// TIA Portal V20 export
FUNCTION_BLOCK "CallInterfaceSignals"   // FB38, LAD
TITLE = CallInterfaceSignals
AUTHOR : SICAR
FAMILY : Diag
VERSION : 1.0
// Der Baustein dient als Aufrufschnittstelle für den Funktionsbaustein „LSicar_InterfaceSignalsBool“. Er ist als Funktionsbaustein ausgeführt, um die intern aufgerufenen FBs mittels Multiinstanzen realisieren zu können.  
// Die Funktionsbausteine und das zugehörige WinCC-Bild sind für 16 Signaldatensätze („Schnittstelle Signale 01“ … „Schnittstellen Signale 16“) mit jeweils 32 boolschen Signalen vorgesehen.  
// 
// **PLC-Datentypen**  
//  LSicar_typeInterfaceSignalsBool 
//  typeInterfaceSignalsHmi 
//  LSicar _typeInterfaceSignals 
// 
// **WinCC-Diagnosebild**  
// 
// ![Icon](_Icon/reference.PNG)
// 
// siehe ..\Library Types\LSicar_InterfaceSignalsBool.pdf  
// 
//  
// 
// **Beispielaufruf**  
// Abbildung in Kontaktplan (KOP).  D:\Software\Symbols_Icons\BMPs-JPGs-PNGs\Verschiedene\symb_user_goto_transparent.pngEin lauffähiger Programm-Aufruf hierzu ist im „SICAR-StartUp“-Projekt enthalten.  
// 
// **Aufrufschnittstelle**  
// Der Baustein wird einmalig im zyklischen Programm aufgerufen.  
// 
// **Intern verwendete „Erweiterte Anweisungen / Bausteine“**  
// ..\Library Types\LSicar_InterfaceSignalsBool.pdf
// The block serves as a calling interface of the block “InterfaceSignalsBool“. The block is designed as function block in order to implement the block calls as multi-instances.
// stored: IsIECCheckEnabled true, MemoryReserve 100, SetENOAutomatically true
   VAR
      statReadValueHmi : Bool;   // HMI: Lese Signalwert / HMI: Read value signal
      statSelectSignalsHmi : USInt := 1;   // HMI: Angewählte Interface Schnittstelle (1..16) / HMI: Selected interface signals (1..16)
      statSelectSignalsOld { ExternalAccessible := 'False'; ExternalVisible := 'False'; ExternalWritable := 'False'} : USInt;   // Altwert: Angewählte Interface Schnittstelle / Old value: Selected interface signals
      statRisEdgeReadName { ExternalAccessible := 'False'; ExternalVisible := 'False'; ExternalWritable := 'False'} : Bool;   // Steigende Flanke / Rising edge
      statPosPulseReadName : Bool;   // Positiver Impuls / Positive pulse
      statInterfaceSignalsHmi : Array[0..99] of "typeInterfaceSignalsHmi";   // HMI: Beschreibung, Wert und Symbolischer Name / HMI: Description, value and symbolic name
      instSignals1Left { S7_SetPoint := 'True'} : "LAF_InterfaceSignalsBool";
      instSignals1Right { S7_SetPoint := 'True'} : "LAF_InterfaceSignalsBool";
      instSignals2Left { S7_SetPoint := 'True'} : "LAF_InterfaceSignalsBool";
      instSignals2Right { S7_SetPoint := 'True'} : "LAF_InterfaceSignalsBool";
      instSignals3Left { S7_SetPoint := 'True'} : "LAF_InterfaceSignalsBool";
      instSignals3Right { S7_SetPoint := 'True'} : "LAF_InterfaceSignalsBool";
      instSignals4Left { S7_SetPoint := 'True'} : "LAF_InterfaceSignalsBool";
      instSignals4Right { S7_SetPoint := 'True'} : "LAF_InterfaceSignalsBool";
      instSignals5Left { S7_SetPoint := 'True'} : "LAF_InterfaceSignalsBool";
      instSignals5Right { S7_SetPoint := 'True'} : "LAF_InterfaceSignalsBool";
      instSignals6Left { S7_SetPoint := 'True'} : "LAF_InterfaceSignalsBool";
      instSignals6Right { S7_SetPoint := 'True'} : "LAF_InterfaceSignalsBool";
      instSignals7Left { S7_SetPoint := 'True'} : "LAF_InterfaceSignalsBool";
      instSignals7Right { S7_SetPoint := 'True'} : "LAF_InterfaceSignalsBool";
      instSignals8Left { S7_SetPoint := 'True'} : "LAF_InterfaceSignalsBool";
      instSignals8Right { S7_SetPoint := 'True'} : "LAF_InterfaceSignalsBool";
      instSignals9Left { S7_SetPoint := 'True'} : "LAF_InterfaceSignalsBool";
      instSignals9Right { S7_SetPoint := 'True'} : "LAF_InterfaceSignalsBool";
      instSignals10Left { S7_SetPoint := 'True'} : "LAF_InterfaceSignalsBool";
      instSignals10Right { S7_SetPoint := 'True'} : "LAF_InterfaceSignalsBool";
      instSignals11Left { S7_SetPoint := 'True'} : "LAF_InterfaceSignalsBool";
      instSignals11Right { S7_SetPoint := 'True'} : "LAF_InterfaceSignalsBool";
      instSignals12Left { S7_SetPoint := 'True'} : "LAF_InterfaceSignalsBool";
      instSignals12Right { S7_SetPoint := 'True'} : "LAF_InterfaceSignalsBool";
      instSignals13Left { S7_SetPoint := 'True'} : "LAF_InterfaceSignalsBool";
      instSignals13Right { S7_SetPoint := 'True'} : "LAF_InterfaceSignalsBool";
      instSignals14Left { S7_SetPoint := 'True'} : "LAF_InterfaceSignalsBool";
      instSignals14Right { S7_SetPoint := 'True'} : "LAF_InterfaceSignalsBool";
      instSignals15Left { S7_SetPoint := 'True'} : "LAF_InterfaceSignalsBool";
      instSignals15Right { S7_SetPoint := 'True'} : "LAF_InterfaceSignalsBool";
      instSignals16Left { S7_SetPoint := 'True'} : "LAF_InterfaceSignalsBool";
      instSignals16Right { S7_SetPoint := 'True'} : "LAF_InterfaceSignalsBool";
      instSignals17Left { S7_SetPoint := 'True'} : "LAF_InterfaceSignalsBool";
      instSignals17Right { S7_SetPoint := 'True'} : "LAF_InterfaceSignalsBool";
      instSignals18Left { S7_SetPoint := 'True'} : "LAF_InterfaceSignalsBool";
      instSignals18Right { S7_SetPoint := 'True'} : "LAF_InterfaceSignalsBool";
      instSignals19Left { S7_SetPoint := 'True'} : "LAF_InterfaceSignalsBool";
      instSignals19Right { S7_SetPoint := 'True'} : "LAF_InterfaceSignalsBool";
      instSignals20Left { S7_SetPoint := 'True'} : "LAF_InterfaceSignalsBool";
      instSignals20Right { S7_SetPoint := 'True'} : "LAF_InterfaceSignalsBool";
      instSignals21Left { S7_SetPoint := 'True'} : "LAF_InterfaceSignalsBool";
      instSignals21Right { S7_SetPoint := 'True'} : "LAF_InterfaceSignalsBool";
      instSignals22Left { S7_SetPoint := 'True'} : "LAF_InterfaceSignalsBool";
      instSignals22Right { S7_SetPoint := 'True'} : "LAF_InterfaceSignalsBool";
      instSignals23Left { S7_SetPoint := 'True'} : "LAF_InterfaceSignalsBool";
      instSignals23Right { S7_SetPoint := 'True'} : "LAF_InterfaceSignalsBool";
      instSignals24Left { S7_SetPoint := 'True'} : "LAF_InterfaceSignalsBool";
      instSignals24Right { S7_SetPoint := 'True'} : "LAF_InterfaceSignalsBool";
      instSignals25Left { S7_SetPoint := 'True'} : "LAF_InterfaceSignalsBool";
      instSignals25Right { S7_SetPoint := 'True'} : "LAF_InterfaceSignalsBool";
      instSignals26Left { S7_SetPoint := 'True'} : "LAF_InterfaceSignalsBool";
      instSignals26Right { S7_SetPoint := 'True'} : "LAF_InterfaceSignalsBool";
      instSignals27Left { S7_SetPoint := 'True'} : "LAF_InterfaceSignalsBool";
      instSignals27Right { S7_SetPoint := 'True'} : "LAF_InterfaceSignalsBool";
      instSignals28Left { S7_SetPoint := 'True'} : "LAF_InterfaceSignalsBool";
      instSignals28Right { S7_SetPoint := 'True'} : "LAF_InterfaceSignalsBool";
      instSignals29Left { S7_SetPoint := 'True'} : "LAF_InterfaceSignalsBool";
      instSignals29Right { S7_SetPoint := 'True'} : "LAF_InterfaceSignalsBool";
      instSignals30Left { S7_SetPoint := 'True'} : "LAF_InterfaceSignalsBool";
      instSignals30Right { S7_SetPoint := 'True'} : "LAF_InterfaceSignalsBool";
      instSignals31Left { S7_SetPoint := 'True'} : "LAF_InterfaceSignalsBool";
      instSignals31Right { S7_SetPoint := 'True'} : "LAF_InterfaceSignalsBool";
      instSignals32Left { S7_SetPoint := 'True'} : "LAF_InterfaceSignalsBool";
      instSignals32Right { S7_SetPoint := 'True'} : "LAF_InterfaceSignalsBool";
      instSignals33Left { S7_SetPoint := 'True'} : "LAF_InterfaceSignalsBool";
      instSignals33Right { S7_SetPoint := 'True'} : "LAF_InterfaceSignalsBool";
      instSignals34Left { S7_SetPoint := 'True'} : "LAF_InterfaceSignalsBool";
      instSignals34Right { S7_SetPoint := 'True'} : "LAF_InterfaceSignalsBool";
      instSignals35Left { S7_SetPoint := 'True'} : "LAF_InterfaceSignalsBool";
      instSignals35Right { S7_SetPoint := 'True'} : "LAF_InterfaceSignalsBool";
      instSignals36Left { S7_SetPoint := 'True'} : "LAF_InterfaceSignalsBool";
      instSignals36Right { S7_SetPoint := 'True'} : "LAF_InterfaceSignalsBool";
      instSignals37Left { S7_SetPoint := 'True'} : "LAF_InterfaceSignalsBool";
      instSignals37Right { S7_SetPoint := 'True'} : "LAF_InterfaceSignalsBool";
      instSignals38Left { S7_SetPoint := 'True'} : "LAF_InterfaceSignalsBool";
      instSignals38Right { S7_SetPoint := 'True'} : "LAF_InterfaceSignalsBool";
      instSignals39Left { S7_SetPoint := 'True'} : "LAF_InterfaceSignalsBool";
      instSignals39Right { S7_SetPoint := 'True'} : "LAF_InterfaceSignalsBool";
      instSignals40Left { S7_SetPoint := 'True'} : "LAF_InterfaceSignalsBool";
      instSignals40Right { S7_SetPoint := 'True'} : "LAF_InterfaceSignalsBool";
      instSignals41Left { S7_SetPoint := 'True'} : "LAF_InterfaceSignalsBool";
      instSignals41Right { S7_SetPoint := 'True'} : "LAF_InterfaceSignalsBool";
      instSignals42Left { S7_SetPoint := 'True'} : "LAF_InterfaceSignalsBool";
      instSignals42Right { S7_SetPoint := 'True'} : "LAF_InterfaceSignalsBool";
      instSignals43Left { S7_SetPoint := 'True'} : "LAF_InterfaceSignalsBool";
      instSignals43Right { S7_SetPoint := 'True'} : "LAF_InterfaceSignalsBool";
      instSignals44Left { S7_SetPoint := 'True'} : "LAF_InterfaceSignalsBool";
      instSignals44Right { S7_SetPoint := 'True'} : "LAF_InterfaceSignalsBool";
      instSignals45Left { S7_SetPoint := 'True'} : "LAF_InterfaceSignalsBool";
      instSignals45Right { S7_SetPoint := 'True'} : "LAF_InterfaceSignalsBool";
      instSignals46Left { S7_SetPoint := 'True'} : "LAF_InterfaceSignalsBool";
      instSignals46Right { S7_SetPoint := 'True'} : "LAF_InterfaceSignalsBool";
      instSignals47Left { S7_SetPoint := 'True'} : "LAF_InterfaceSignalsBool";
      instSignals47Right { S7_SetPoint := 'True'} : "LAF_InterfaceSignalsBool";
      instSignals48Left { S7_SetPoint := 'True'} : "LAF_InterfaceSignalsBool";
      instSignals48Right { S7_SetPoint := 'True'} : "LAF_InterfaceSignalsBool";
      instSignals49Left { S7_SetPoint := 'True'} : "LAF_InterfaceSignalsBool";
      instSignals49Right { S7_SetPoint := 'True'} : "LAF_InterfaceSignalsBool";
      instSignals50Left { S7_SetPoint := 'True'} : "LAF_InterfaceSignalsBool";
      instSignals50Right { S7_SetPoint := 'True'} : "LAF_InterfaceSignalsBool";
      instSignals51Left { S7_SetPoint := 'True'} : "LAF_InterfaceSignalsBool";
      instSignals51Right { S7_SetPoint := 'True'} : "LAF_InterfaceSignalsBool";
      instSignals52Left { S7_SetPoint := 'True'} : "LAF_InterfaceSignalsBool";
      instSignals52Right { S7_SetPoint := 'True'} : "LAF_InterfaceSignalsBool";
      instSignals53Left { S7_SetPoint := 'True'} : "LAF_InterfaceSignalsBool";
      instSignals53Right { S7_SetPoint := 'True'} : "LAF_InterfaceSignalsBool";
      instSignals54Left { S7_SetPoint := 'True'} : "LAF_InterfaceSignalsBool";
      instSignals54Right { S7_SetPoint := 'True'} : "LAF_InterfaceSignalsBool";
      instSignals55Left { S7_SetPoint := 'True'} : "LAF_InterfaceSignalsBool";
      instSignals55Right { S7_SetPoint := 'True'} : "LAF_InterfaceSignalsBool";
      instSignals56Left { S7_SetPoint := 'True'} : "LAF_InterfaceSignalsBool";
      instSignals56Right { S7_SetPoint := 'True'} : "LAF_InterfaceSignalsBool";
      instSignals57Left { S7_SetPoint := 'True'} : "LAF_InterfaceSignalsBool";
      instSignals57Right { S7_SetPoint := 'True'} : "LAF_InterfaceSignalsBool";
      instSignals58Left { S7_SetPoint := 'True'} : "LAF_InterfaceSignalsBool";
      instSignals58Right { S7_SetPoint := 'True'} : "LAF_InterfaceSignalsBool";
      instSignals59Left { S7_SetPoint := 'True'} : "LAF_InterfaceSignalsBool";
      instSignals59Right { S7_SetPoint := 'True'} : "LAF_InterfaceSignalsBool";
      instSignals60Left { S7_SetPoint := 'True'} : "LAF_InterfaceSignalsBool";
      instSignals60Right { S7_SetPoint := 'True'} : "LAF_InterfaceSignalsBool";
      instSignals61Left { S7_SetPoint := 'True'} : "LAF_InterfaceSignalsBool";
      instSignals61Right { S7_SetPoint := 'True'} : "LAF_InterfaceSignalsBool";
      instSignals62Left { S7_SetPoint := 'True'} : "LAF_InterfaceSignalsBool";
      instSignals62Right { S7_SetPoint := 'True'} : "LAF_InterfaceSignalsBool";
      instSignals63Left { S7_SetPoint := 'True'} : "LAF_InterfaceSignalsBool";
      instSignals63Right { S7_SetPoint := 'True'} : "LAF_InterfaceSignalsBool";
      instSignals64Left { S7_SetPoint := 'True'} : "LAF_InterfaceSignalsBool";
      instSignals64Right { S7_SetPoint := 'True'} : "LAF_InterfaceSignalsBool";
      instSignals65Left { S7_SetPoint := 'True'} : "LAF_InterfaceSignalsBool";
      instSignals65Right { S7_SetPoint := 'True'} : "LAF_InterfaceSignalsBool";
      instSignals66Left { S7_SetPoint := 'True'} : "LAF_InterfaceSignalsBool";
      instSignals66Right { S7_SetPoint := 'True'} : "LAF_InterfaceSignalsBool";
      instSignals67Left { S7_SetPoint := 'True'} : "LAF_InterfaceSignalsBool";
      instSignals67Right { S7_SetPoint := 'True'} : "LAF_InterfaceSignalsBool";
      instSignals68Left { S7_SetPoint := 'True'} : "LAF_InterfaceSignalsBool";
      instSignals68Right { S7_SetPoint := 'True'} : "LAF_InterfaceSignalsBool";
      instSignals69Left { S7_SetPoint := 'True'} : "LAF_InterfaceSignalsBool";
      instSignals69Right { S7_SetPoint := 'True'} : "LAF_InterfaceSignalsBool";
      instSignals70Left { S7_SetPoint := 'True'} : "LAF_InterfaceSignalsBool";
      instSignals70Right { S7_SetPoint := 'True'} : "LAF_InterfaceSignalsBool";
      instSignals71Left { S7_SetPoint := 'True'} : "LAF_InterfaceSignalsBool";
      instSignals71Right { S7_SetPoint := 'True'} : "LAF_InterfaceSignalsBool";
      instSignals72Left { S7_SetPoint := 'True'} : "LAF_InterfaceSignalsBool";
      instSignals72Right { S7_SetPoint := 'True'} : "LAF_InterfaceSignalsBool";
      instSignals73Left { S7_SetPoint := 'True'} : "LAF_InterfaceSignalsBool";
      instSignals73Right { S7_SetPoint := 'True'} : "LAF_InterfaceSignalsBool";
      instSignals74Left { S7_SetPoint := 'True'} : "LAF_InterfaceSignalsBool";
      instSignals74Right { S7_SetPoint := 'True'} : "LAF_InterfaceSignalsBool";
      instSignals75Left { S7_SetPoint := 'True'} : "LAF_InterfaceSignalsBool";
      instSignals75Right { S7_SetPoint := 'True'} : "LAF_InterfaceSignalsBool";
      instSignals76Left { S7_SetPoint := 'True'} : "LAF_InterfaceSignalsBool";
      instSignals76Right { S7_SetPoint := 'True'} : "LAF_InterfaceSignalsBool";
      instSignals77Left { S7_SetPoint := 'True'} : "LAF_InterfaceSignalsBool";
      instSignals77Right { S7_SetPoint := 'True'} : "LAF_InterfaceSignalsBool";
      instSignals78Left { S7_SetPoint := 'True'} : "LAF_InterfaceSignalsBool";
      instSignals78Right { S7_SetPoint := 'True'} : "LAF_InterfaceSignalsBool";
      instSignals79Left { S7_SetPoint := 'True'} : "LAF_InterfaceSignalsBool";
      instSignals79Right { S7_SetPoint := 'True'} : "LAF_InterfaceSignalsBool";
      instSignals80Left { S7_SetPoint := 'True'} : "LAF_InterfaceSignalsBool";
      instSignals80Right { S7_SetPoint := 'True'} : "LAF_InterfaceSignalsBool";
      instSignals81Left { S7_SetPoint := 'True'} : "LAF_InterfaceSignalsBool";
      instSignals81Right { S7_SetPoint := 'True'} : "LAF_InterfaceSignalsBool";
      instSignals82Left { S7_SetPoint := 'True'} : "LAF_InterfaceSignalsBool";
      instSignals82Right { S7_SetPoint := 'True'} : "LAF_InterfaceSignalsBool";
      instSignals83Left { S7_SetPoint := 'True'} : "LAF_InterfaceSignalsBool";
      instSignals83Right { S7_SetPoint := 'True'} : "LAF_InterfaceSignalsBool";
      instSignals84Left { S7_SetPoint := 'True'} : "LAF_InterfaceSignalsBool";
      instSignals84Right { S7_SetPoint := 'True'} : "LAF_InterfaceSignalsBool";
      instSignals85Left { S7_SetPoint := 'True'} : "LAF_InterfaceSignalsBool";
      instSignals85Right { S7_SetPoint := 'True'} : "LAF_InterfaceSignalsBool";
      instSignals86Left { S7_SetPoint := 'True'} : "LAF_InterfaceSignalsBool";
      instSignals86Right { S7_SetPoint := 'True'} : "LAF_InterfaceSignalsBool";
      instSignals87Left { S7_SetPoint := 'True'} : "LAF_InterfaceSignalsBool";
      instSignals87Right { S7_SetPoint := 'True'} : "LAF_InterfaceSignalsBool";
      instSignals88Left { S7_SetPoint := 'True'} : "LAF_InterfaceSignalsBool";
      instSignals88Right { S7_SetPoint := 'True'} : "LAF_InterfaceSignalsBool";
      instSignals89Left { S7_SetPoint := 'True'} : "LAF_InterfaceSignalsBool";
      instSignals89Right { S7_SetPoint := 'True'} : "LAF_InterfaceSignalsBool";
      instSignals90Left { S7_SetPoint := 'True'} : "LAF_InterfaceSignalsBool";
      instSignals90Right { S7_SetPoint := 'True'} : "LAF_InterfaceSignalsBool";
      instSignals91Left { S7_SetPoint := 'True'} : "LAF_InterfaceSignalsBool";
      instSignals91Right { S7_SetPoint := 'True'} : "LAF_InterfaceSignalsBool";
      instSignals92Left { S7_SetPoint := 'True'} : "LAF_InterfaceSignalsBool";
      instSignals92Right { S7_SetPoint := 'True'} : "LAF_InterfaceSignalsBool";
      instSignals93Left { S7_SetPoint := 'True'} : "LAF_InterfaceSignalsBool";
      instSignals93Right { S7_SetPoint := 'True'} : "LAF_InterfaceSignalsBool";
      instSignals94Left { S7_SetPoint := 'True'} : "LAF_InterfaceSignalsBool";
      instSignals94Right { S7_SetPoint := 'True'} : "LAF_InterfaceSignalsBool";
      instSignals95Left { S7_SetPoint := 'True'} : "LAF_InterfaceSignalsBool";
      instSignals95Right { S7_SetPoint := 'True'} : "LAF_InterfaceSignalsBool";
      instSignals96Left { S7_SetPoint := 'True'} : "LAF_InterfaceSignalsBool";
      instSignals96Right { S7_SetPoint := 'True'} : "LAF_InterfaceSignalsBool";
      instSignals97Left { S7_SetPoint := 'True'} : "LAF_InterfaceSignalsBool";
      instSignals97Right { S7_SetPoint := 'True'} : "LAF_InterfaceSignalsBool";
      instSignals98Left { S7_SetPoint := 'True'} : "LAF_InterfaceSignalsBool";
      instSignals98Right { S7_SetPoint := 'True'} : "LAF_InterfaceSignalsBool";
      instSignals99Left { S7_SetPoint := 'True'} : "LAF_InterfaceSignalsBool";
      instSignals99Right { S7_SetPoint := 'True'} : "LAF_InterfaceSignalsBool";
   END_VAR
   VAR_TEMP
      tempLoopCounter : DInt;   // temp. Schleifenzähler / temp. Loop Counter
   END_VAR
   VAR_TEMP   // added for the SCL form of the ladder/FBD networks
      _w1 : Bool;
   END_VAR
BEGIN

REGION Network 1: Beschreibung / BLOCK INFO HEADER
   // **Betriebsart Automatik / Hand**  
   // Der Baustein ist keiner Betriebsart / Betriebsartenbereich zugeordnet.  
   // 
   // **Alarme**  
   // Der Baustein generiert keine Alarme.  
   // 
   // #### PLC-Datentypen  
   // Verwendete PLC-Datentypen für den SPS-Programmbaustein und das zugehörige WinCC-Bild.  
   // 
   // {.pageWidth}
   // ![Image](CallInterfaceSignals/de/image1.PNG)
   //  
   //  
   // #### Bausteinaufrufe 
   // Der Baustein “LSicar_InterfaceSignalsBool“ wird in diesem FB als Multi-Instanz aufgerufen, entspr. nebenstehender beispielhafter Darstellung.  
   // 
   // {.pageWidth}
   // ![Image](CallInterfaceSignals/de/image2.PNG)
   //  
   // Um einen neuen FB aufzurufen, ziehen Sie den FB in ein neues Netzwerk, wählen Sie „Multiinstanz“ aus, vergeben Sie einen Namen und parametrieren Sie den FB-Aufruf.  
   // 
   // {.pageWidth}
   // ![Image](CallInterfaceSignals/de/image3.PNG)
   //  
   //  
   // #### Weitere Hinweise 
   // 
   // #### Updateinfo 
   // 
   // #### Weitere Dokumente 
   // 
   // ![Icon](_Icon/reference.PNG)
   // 
   // ..\Library Types\LSicar_InterfaceSignalsBool.pdf
   // SIEMENS AG / (c)Copyright 2023
   // ------------------------------------------------------------------------------
   // Title:            CallInterfaceSignals (FB38)
   // Comment/Function: The block serves as a calling interface of the block “InterfaceSignalsBool“. The block is designed as function block in order to implement the block calls as multi-instances. 
   // Library/Family:   Diag
   // Author:           SICAR
   // Tested with:      ---
   // Engineering:      TIA Portal V19
   // Restrictions:     -
   // Requirements:     ---
   // ------------------------------------------------------------------------------
   // Change log table:
   // Version  | Date       | Expert in charge       | Changes applied
   // ---------|------------|------------------------|------------------------------
   // 01.00.00 | 11.12.2023 | SICAR
   //                         First released version
END_REGION

REGION Network 2: DESCRIPTION
   // Function block and corresponding WinCC screen are prepared for 16 data sets (“InterfaceSignals01“ through .”InterfaceSignals16“) with 32 Boolean signals each.  
   // 
   // **PLC-Data types**   
   // 
   // * LSicar_typeInterfaceSignalsBool 
   // * LSicar _typeInterfaceSignals 
   // * typeInterfaceSignalsHmi 
   // 
   // **WinCC-Faceplate**  
   // 
   // <None> 
   // 
   // **WinCC Diagnostic screen**   
   // 
   // See: ..\Library Types\LSicar_InterfaceSignalsBool.pdf  
   // 
   // **Block call example** 
   // 
   // View in ladder-logic (LAD), without parameter settings.  
   // An executable program call is available in the “SICAR-Startup” project.  
   // 
   // **Calling interface**  
   // 
   // The block is be called once in the cyclic program.  
   // 
   // **Internally used „Extended instructions / blocks“**  
   // 
   // See: ..\Library Types\LSicar_InterfaceSignalsBool.pdf
END_REGION

REGION Network 3: Initialisierung Loop_1 / Initialization Loop_1
   // Vorbesetzen des Schleifenindex / Preset the loop index
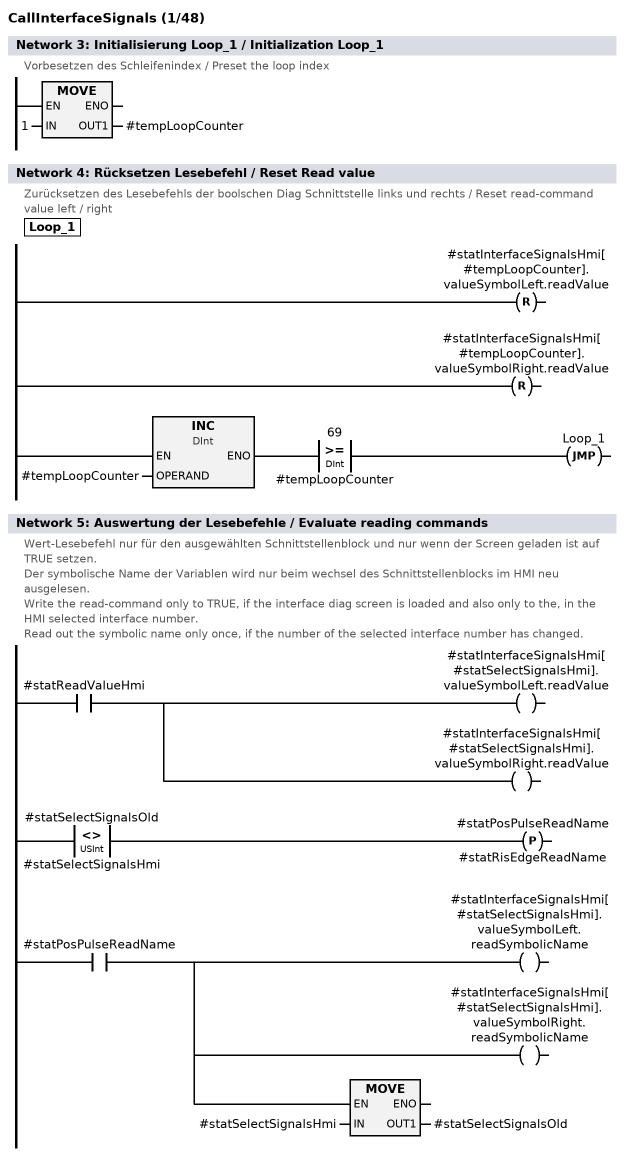
   RUNG wire#powerrail
      Move(in := 1, out1 => #tempLoopCounter)
   END_RUNG
   // the same network as SCL:
   #tempLoopCounter := 1;
END_REGION

REGION Network 4: Rücksetzen Lesebefehl / Reset Read value
   // Zurücksetzen des Lesebefehls der boolschen Diag Schnittstelle links und rechts / Reset read-command value left / right
   Label( Loop_1 )
   RUNG wire#powerrail
      R_Coil( #statInterfaceSignalsHmi[#tempLoopCounter].valueSymbolLeft.readValue )
   END_RUNG
   RUNG wire#powerrail
      R_Coil( #statInterfaceSignalsHmi[#tempLoopCounter].valueSymbolRight.readValue )
   END_RUNG
   RUNG wire#powerrail
      { S7_Templates := "DestType := DInt" } Inc( #tempLoopCounter )
      { S7_Templates := "SrcType := DInt" } GE_Contact(in1 := 69, in2 := #tempLoopCounter)
      JumpCoil( Loop_1 )
   END_RUNG
   // the same network as SCL:
   Loop_1:
   #statInterfaceSignalsHmi[#tempLoopCounter].valueSymbolLeft.readValue := FALSE;
   #statInterfaceSignalsHmi[#tempLoopCounter].valueSymbolRight.readValue := FALSE;
   #tempLoopCounter := #tempLoopCounter + 1;
   IF 69 >= #tempLoopCounter THEN GOTO Loop_1; END_IF;
END_REGION

REGION Network 5: Auswertung der Lesebefehle / Evaluate reading commands
   // Wert-Lesebefehl nur für den ausgewählten Schnittstellenblock und nur wenn der Screen geladen ist auf TRUE setzen.
   // Der symbolische Name der Variablen wird nur beim wechsel des Schnittstellenblocks im HMI neu ausgelesen.
   // Write the read-command only to TRUE, if the interface diag screen is loaded and also only to the, in the HMI selected interface number.
   // Read out the symbolic name only once, if the number of the selected interface number has changed.
   #statInterfaceSignalsHmi[#statSelectSignalsHmi].valueSymbolLeft.readValue := #statReadValueHmi;
   #statInterfaceSignalsHmi[#statSelectSignalsHmi].valueSymbolRight.readValue := #statReadValueHmi;
   #_w1 := #statSelectSignalsOld <> #statSelectSignalsHmi;
   #statPosPulseReadName := #_w1 AND NOT #statRisEdgeReadName;   // rising edge
   #statRisEdgeReadName := #_w1;
   #statInterfaceSignalsHmi[#statSelectSignalsHmi].valueSymbolLeft.readSymbolicName := #statPosPulseReadName;
   #statInterfaceSignalsHmi[#statSelectSignalsHmi].valueSymbolRight.readSymbolicName := #statPosPulseReadName;
   IF #statPosPulseReadName THEN #statSelectSignalsOld := #statSelectSignalsHmi; END_IF;
END_REGION

REGION Network 6: Interface Signals 03 -Example: System flags & Clock flags- / Interface Signals 01
   // Aufruf des Schnittstellen Signal Bausteins für die Systemvariablen / Call the interface signals bool blocks of system tags
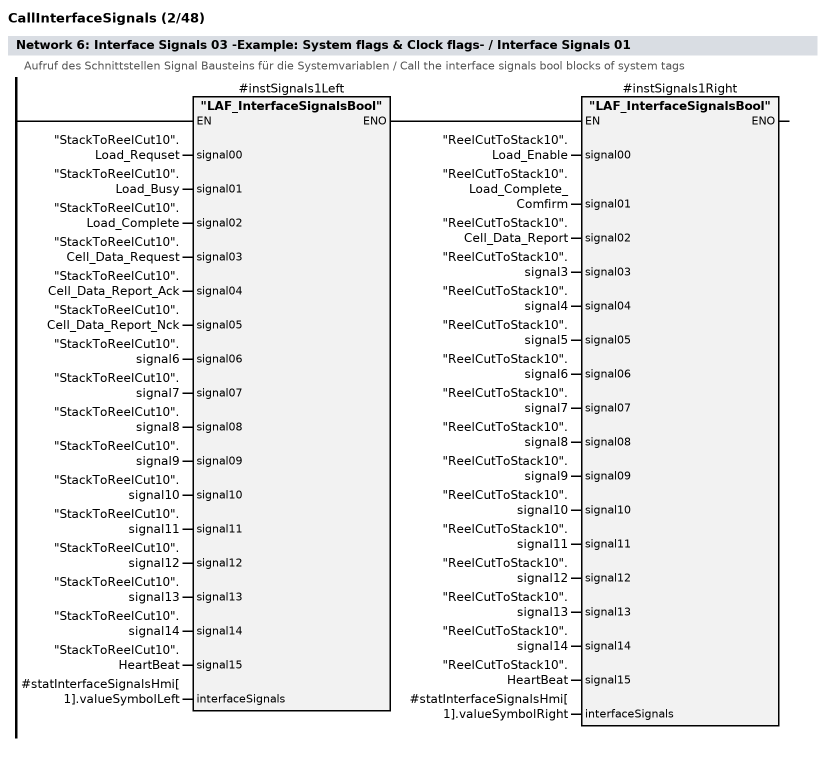
   RUNG wire#powerrail
      #instSignals1Left(signal00 := "StackToReelCut10".Load_Requset, signal01 := "StackToReelCut10".Load_Busy, signal02 := "StackToReelCut10".Load_Complete, signal03 := "StackToReelCut10".Cell_Data_Request, signal04 := "StackToReelCut10".Cell_Data_Report_Ack, signal05 := "StackToReelCut10".Cell_Data_Report_Nck, signal06 := "StackToReelCut10".signal6, signal07 := "StackToReelCut10".signal7, signal08 := "StackToReelCut10".signal8, signal09 := "StackToReelCut10".signal9, signal10 := "StackToReelCut10".signal10, signal11 := "StackToReelCut10".signal11, signal12 := "StackToReelCut10".signal12, signal13 := "StackToReelCut10".signal13, signal14 := "StackToReelCut10".signal14, signal15 := "StackToReelCut10".HeartBeat, interfaceSignals := #statInterfaceSignalsHmi[1].valueSymbolLeft)
      #instSignals1Right(signal00 := "ReelCutToStack10".Load_Enable, signal01 := "ReelCutToStack10".Load_Complete_Comfirm, signal02 := "ReelCutToStack10".Cell_Data_Report, signal03 := "ReelCutToStack10".signal3, signal04 := "ReelCutToStack10".signal4, signal05 := "ReelCutToStack10".signal5, signal06 := "ReelCutToStack10".signal6, signal07 := "ReelCutToStack10".signal7, signal08 := "ReelCutToStack10".signal8, signal09 := "ReelCutToStack10".signal9, signal10 := "ReelCutToStack10".signal10, signal11 := "ReelCutToStack10".signal11, signal12 := "ReelCutToStack10".signal12, signal13 := "ReelCutToStack10".signal13, signal14 := "ReelCutToStack10".signal14, signal15 := "ReelCutToStack10".HeartBeat, interfaceSignals := #statInterfaceSignalsHmi[1].valueSymbolRight)
   END_RUNG
   // the same network as SCL:
   #instSignals1Left(signal00 := "StackToReelCut10".Load_Requset,   // "LAF_InterfaceSignalsBool"
                     signal01 := "StackToReelCut10".Load_Busy,
                     signal02 := "StackToReelCut10".Load_Complete,
                     signal03 := "StackToReelCut10".Cell_Data_Request,
                     signal04 := "StackToReelCut10".Cell_Data_Report_Ack,
                     signal05 := "StackToReelCut10".Cell_Data_Report_Nck,
                     signal06 := "StackToReelCut10".signal6,
                     signal07 := "StackToReelCut10".signal7,
                     signal08 := "StackToReelCut10".signal8,
                     signal09 := "StackToReelCut10".signal9,
                     signal10 := "StackToReelCut10".signal10,
                     signal11 := "StackToReelCut10".signal11,
                     signal12 := "StackToReelCut10".signal12,
                     signal13 := "StackToReelCut10".signal13,
                     signal14 := "StackToReelCut10".signal14,
                     signal15 := "StackToReelCut10".HeartBeat,
                     interfaceSignals := #statInterfaceSignalsHmi[1].valueSymbolLeft,
                     ENO => #_w1);
   IF #_w1 THEN
       #instSignals1Right(signal00 := "ReelCutToStack10".Load_Enable,   // "LAF_InterfaceSignalsBool"
                          signal01 := "ReelCutToStack10".Load_Complete_Comfirm,
                          signal02 := "ReelCutToStack10".Cell_Data_Report,
                          signal03 := "ReelCutToStack10".signal3,
                          signal04 := "ReelCutToStack10".signal4,
                          signal05 := "ReelCutToStack10".signal5,
                          signal06 := "ReelCutToStack10".signal6,
                          signal07 := "ReelCutToStack10".signal7,
                          signal08 := "ReelCutToStack10".signal8,
                          signal09 := "ReelCutToStack10".signal9,
                          signal10 := "ReelCutToStack10".signal10,
                          signal11 := "ReelCutToStack10".signal11,
                          signal12 := "ReelCutToStack10".signal12,
                          signal13 := "ReelCutToStack10".signal13,
                          signal14 := "ReelCutToStack10".signal14,
                          signal15 := "ReelCutToStack10".HeartBeat,
                          interfaceSignals := #statInterfaceSignalsHmi[1].valueSymbolRight);
   END_IF;
END_REGION

REGION Network 7: Interface Signals 03 -Example: System flags & Clock flags- / Interface Signals 02
   // Aufruf des Schnittstellen Signal Bausteins für die Systemvariablen / Call the interface signals bool blocks of system tags
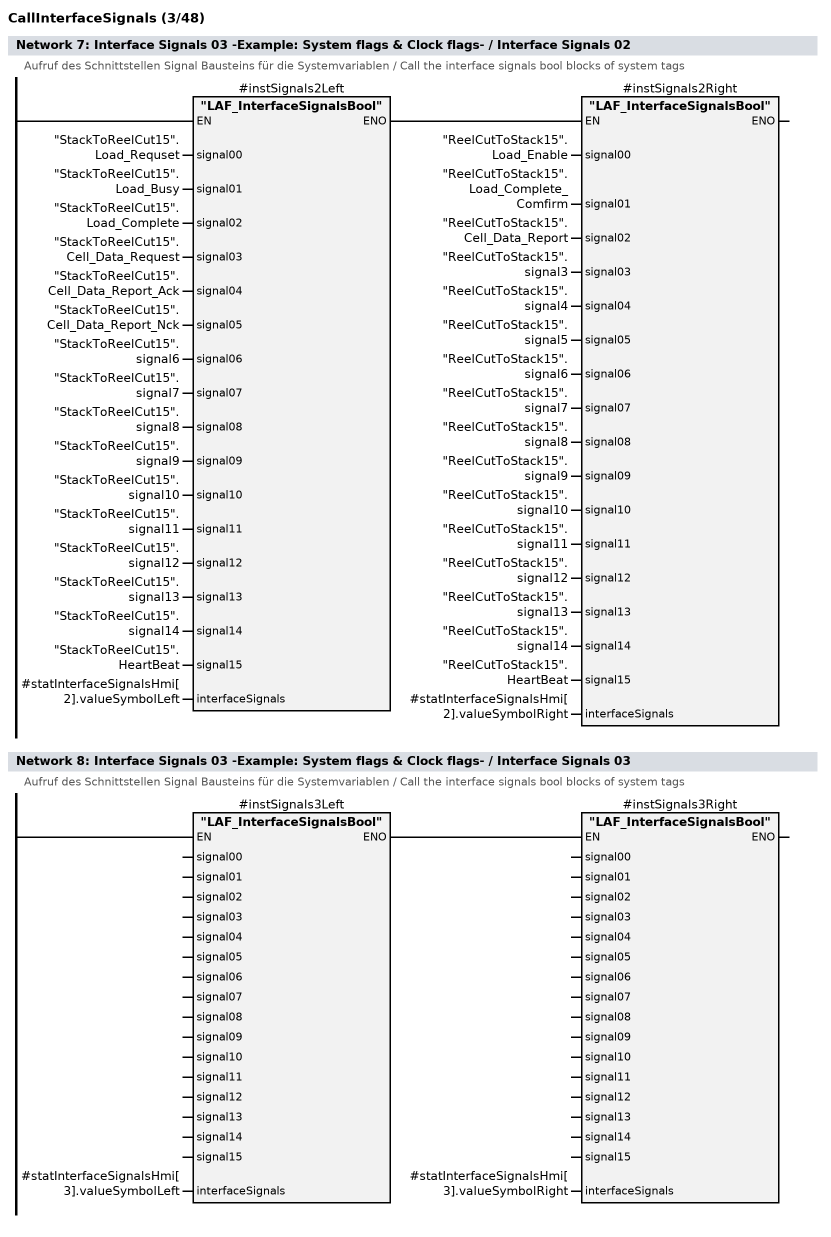
   RUNG wire#powerrail
      #instSignals2Left(signal00 := "StackToReelCut15".Load_Requset, signal01 := "StackToReelCut15".Load_Busy, signal02 := "StackToReelCut15".Load_Complete, signal03 := "StackToReelCut15".Cell_Data_Request, signal04 := "StackToReelCut15".Cell_Data_Report_Ack, signal05 := "StackToReelCut15".Cell_Data_Report_Nck, signal06 := "StackToReelCut15".signal6, signal07 := "StackToReelCut15".signal7, signal08 := "StackToReelCut15".signal8, signal09 := "StackToReelCut15".signal9, signal10 := "StackToReelCut15".signal10, signal11 := "StackToReelCut15".signal11, signal12 := "StackToReelCut15".signal12, signal13 := "StackToReelCut15".signal13, signal14 := "StackToReelCut15".signal14, signal15 := "StackToReelCut15".HeartBeat, interfaceSignals := #statInterfaceSignalsHmi[2].valueSymbolLeft)
      #instSignals2Right(signal00 := "ReelCutToStack15".Load_Enable, signal01 := "ReelCutToStack15".Load_Complete_Comfirm, signal02 := "ReelCutToStack15".Cell_Data_Report, signal03 := "ReelCutToStack15".signal3, signal04 := "ReelCutToStack15".signal4, signal05 := "ReelCutToStack15".signal5, signal06 := "ReelCutToStack15".signal6, signal07 := "ReelCutToStack15".signal7, signal08 := "ReelCutToStack15".signal8, signal09 := "ReelCutToStack15".signal9, signal10 := "ReelCutToStack15".signal10, signal11 := "ReelCutToStack15".signal11, signal12 := "ReelCutToStack15".signal12, signal13 := "ReelCutToStack15".signal13, signal14 := "ReelCutToStack15".signal14, signal15 := "ReelCutToStack15".HeartBeat, interfaceSignals := #statInterfaceSignalsHmi[2].valueSymbolRight)
   END_RUNG
   // the same network as SCL:
   #instSignals2Left(signal00 := "StackToReelCut15".Load_Requset,   // "LAF_InterfaceSignalsBool"
                     signal01 := "StackToReelCut15".Load_Busy,
                     signal02 := "StackToReelCut15".Load_Complete,
                     signal03 := "StackToReelCut15".Cell_Data_Request,
                     signal04 := "StackToReelCut15".Cell_Data_Report_Ack,
                     signal05 := "StackToReelCut15".Cell_Data_Report_Nck,
                     signal06 := "StackToReelCut15".signal6,
                     signal07 := "StackToReelCut15".signal7,
                     signal08 := "StackToReelCut15".signal8,
                     signal09 := "StackToReelCut15".signal9,
                     signal10 := "StackToReelCut15".signal10,
                     signal11 := "StackToReelCut15".signal11,
                     signal12 := "StackToReelCut15".signal12,
                     signal13 := "StackToReelCut15".signal13,
                     signal14 := "StackToReelCut15".signal14,
                     signal15 := "StackToReelCut15".HeartBeat,
                     interfaceSignals := #statInterfaceSignalsHmi[2].valueSymbolLeft,
                     ENO => #_w1);
   IF #_w1 THEN
       #instSignals2Right(signal00 := "ReelCutToStack15".Load_Enable,   // "LAF_InterfaceSignalsBool"
                          signal01 := "ReelCutToStack15".Load_Complete_Comfirm,
                          signal02 := "ReelCutToStack15".Cell_Data_Report,
                          signal03 := "ReelCutToStack15".signal3,
                          signal04 := "ReelCutToStack15".signal4,
                          signal05 := "ReelCutToStack15".signal5,
                          signal06 := "ReelCutToStack15".signal6,
                          signal07 := "ReelCutToStack15".signal7,
                          signal08 := "ReelCutToStack15".signal8,
                          signal09 := "ReelCutToStack15".signal9,
                          signal10 := "ReelCutToStack15".signal10,
                          signal11 := "ReelCutToStack15".signal11,
                          signal12 := "ReelCutToStack15".signal12,
                          signal13 := "ReelCutToStack15".signal13,
                          signal14 := "ReelCutToStack15".signal14,
                          signal15 := "ReelCutToStack15".HeartBeat,
                          interfaceSignals := #statInterfaceSignalsHmi[2].valueSymbolRight);
   END_IF;
END_REGION

REGION Network 8: Interface Signals 03 -Example: System flags & Clock flags- / Interface Signals 03
   // Aufruf des Schnittstellen Signal Bausteins für die Systemvariablen / Call the interface signals bool blocks of system tags
   RUNG wire#powerrail
      #instSignals3Left(signal00 :=, signal01 :=, signal02 :=, signal03 :=, signal04 :=, signal05 :=, signal06 :=, signal07 :=, signal08 :=, signal09 :=, signal10 :=, signal11 :=, signal12 :=, signal13 :=, signal14 :=, signal15 :=, interfaceSignals := #statInterfaceSignalsHmi[3].valueSymbolLeft)
      #instSignals3Right(signal00 :=, signal01 :=, signal02 :=, signal03 :=, signal04 :=, signal05 :=, signal06 :=, signal07 :=, signal08 :=, signal09 :=, signal10 :=, signal11 :=, signal12 :=, signal13 :=, signal14 :=, signal15 :=, interfaceSignals := #statInterfaceSignalsHmi[3].valueSymbolRight)
   END_RUNG
   // the same network as SCL:
   #instSignals3Left(interfaceSignals := #statInterfaceSignalsHmi[3].valueSymbolLeft, ENO => #_w1);   // "LAF_InterfaceSignalsBool"
   IF #_w1 THEN
       #instSignals3Right(interfaceSignals := #statInterfaceSignalsHmi[3].valueSymbolRight);   // "LAF_InterfaceSignalsBool"
   END_IF;
END_REGION

REGION Network 9: Interface Signals 04 -Example: Model Flex-Pro-Line - IN/OUT- / Interface Signals 04
   // Aufruf des Schnittstellen Signal Bausteins Ba-Bereich 4 / Call the interface signals bool blocks of opmode 4
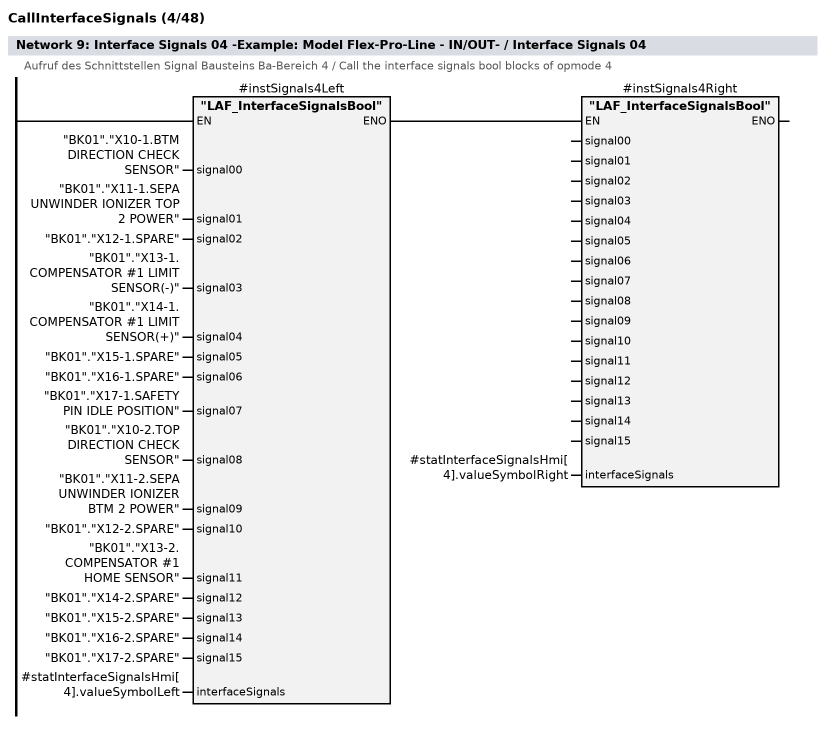
   RUNG wire#powerrail
      #instSignals4Left(signal00 := "BK01"."X10-1.BTM DIRECTION CHECK SENSOR", signal01 := "BK01"."X11-1.SEPA UNWINDER IONIZER TOP 2 POWER", signal02 := "BK01"."X12-1.SPARE", signal03 := "BK01"."X13-1.COMPENSATOR #1 LIMIT SENSOR(-)", signal04 := "BK01"."X14-1.COMPENSATOR #1 LIMIT SENSOR(+)", signal05 := "BK01"."X15-1.SPARE", signal06 := "BK01"."X16-1.SPARE", signal07 := "BK01"."X17-1.SAFETY PIN IDLE POSITION", signal08 := "BK01"."X10-2.TOP DIRECTION CHECK SENSOR", signal09 := "BK01"."X11-2.SEPA UNWINDER IONIZER BTM 2 POWER", signal10 := "BK01"."X12-2.SPARE", signal11 := "BK01"."X13-2.COMPENSATOR #1 HOME SENSOR", signal12 := "BK01"."X14-2.SPARE", signal13 := "BK01"."X15-2.SPARE", signal14 := "BK01"."X16-2.SPARE", signal15 := "BK01"."X17-2.SPARE", interfaceSignals := #statInterfaceSignalsHmi[4].valueSymbolLeft)
      #instSignals4Right(signal00 :=, signal01 :=, signal02 :=, signal03 :=, signal04 :=, signal05 :=, signal06 :=, signal07 :=, signal08 :=, signal09 :=, signal10 :=, signal11 :=, signal12 :=, signal13 :=, signal14 :=, signal15 :=, interfaceSignals := #statInterfaceSignalsHmi[4].valueSymbolRight)
   END_RUNG
   // the same network as SCL:
   #instSignals4Left(signal00 := "BK01"."X10-1.BTM DIRECTION CHECK SENSOR",   // "LAF_InterfaceSignalsBool"
                     signal01 := "BK01"."X11-1.SEPA UNWINDER IONIZER TOP 2 POWER",
                     signal02 := "BK01"."X12-1.SPARE",
                     signal03 := "BK01"."X13-1.COMPENSATOR #1 LIMIT SENSOR(-)",
                     signal04 := "BK01"."X14-1.COMPENSATOR #1 LIMIT SENSOR(+)",
                     signal05 := "BK01"."X15-1.SPARE",
                     signal06 := "BK01"."X16-1.SPARE",
                     signal07 := "BK01"."X17-1.SAFETY PIN IDLE POSITION",
                     signal08 := "BK01"."X10-2.TOP DIRECTION CHECK SENSOR",
                     signal09 := "BK01"."X11-2.SEPA UNWINDER IONIZER BTM 2 POWER",
                     signal10 := "BK01"."X12-2.SPARE",
                     signal11 := "BK01"."X13-2.COMPENSATOR #1 HOME SENSOR",
                     signal12 := "BK01"."X14-2.SPARE",
                     signal13 := "BK01"."X15-2.SPARE",
                     signal14 := "BK01"."X16-2.SPARE",
                     signal15 := "BK01"."X17-2.SPARE",
                     interfaceSignals := #statInterfaceSignalsHmi[4].valueSymbolLeft,
                     ENO => #_w1);
   IF #_w1 THEN
       #instSignals4Right(interfaceSignals := #statInterfaceSignalsHmi[4].valueSymbolRight);   // "LAF_InterfaceSignalsBool"
   END_IF;
END_REGION

REGION Network 10: Interface Signals 05 -Example: Model Flex-Pro-Line - IN/OUT- / Interface Signals 05
   // Aufruf des Schnittstellen Signal Bausteins Ba-Bereich 4 / Call the interface signals bool blocks of opmode 4
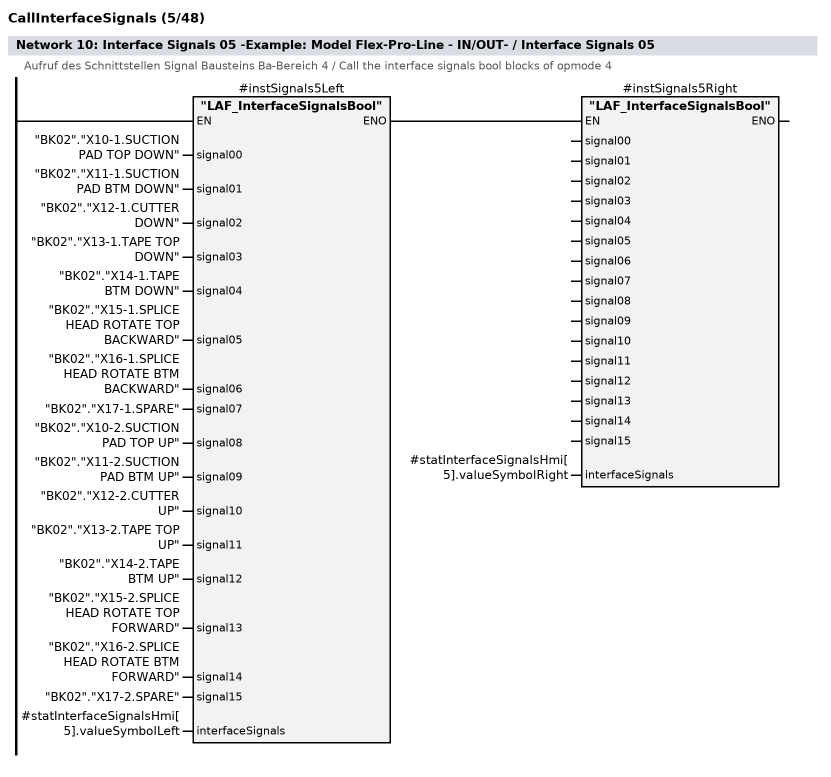
   RUNG wire#powerrail
      #instSignals5Left(signal00 := "BK02"."X10-1.SUCTION PAD TOP DOWN", signal01 := "BK02"."X11-1.SUCTION PAD BTM DOWN", signal02 := "BK02"."X12-1.CUTTER DOWN", signal03 := "BK02"."X13-1.TAPE TOP DOWN", signal04 := "BK02"."X14-1.TAPE BTM DOWN", signal05 := "BK02"."X15-1.SPLICE HEAD ROTATE TOP BACKWARD", signal06 := "BK02"."X16-1.SPLICE HEAD ROTATE BTM BACKWARD", signal07 := "BK02"."X17-1.SPARE", signal08 := "BK02"."X10-2.SUCTION PAD TOP UP", signal09 := "BK02"."X11-2.SUCTION PAD BTM UP", signal10 := "BK02"."X12-2.CUTTER UP", signal11 := "BK02"."X13-2.TAPE TOP UP", signal12 := "BK02"."X14-2.TAPE BTM UP", signal13 := "BK02"."X15-2.SPLICE HEAD ROTATE TOP FORWARD", signal14 := "BK02"."X16-2.SPLICE HEAD ROTATE BTM FORWARD", signal15 := "BK02"."X17-2.SPARE", interfaceSignals := #statInterfaceSignalsHmi[5].valueSymbolLeft)
      #instSignals5Right(signal00 :=, signal01 :=, signal02 :=, signal03 :=, signal04 :=, signal05 :=, signal06 :=, signal07 :=, signal08 :=, signal09 :=, signal10 :=, signal11 :=, signal12 :=, signal13 :=, signal14 :=, signal15 :=, interfaceSignals := #statInterfaceSignalsHmi[5].valueSymbolRight)
   END_RUNG
   // the same network as SCL:
   #instSignals5Left(signal00 := "BK02"."X10-1.SUCTION PAD TOP DOWN",   // "LAF_InterfaceSignalsBool"
                     signal01 := "BK02"."X11-1.SUCTION PAD BTM DOWN",
                     signal02 := "BK02"."X12-1.CUTTER DOWN",
                     signal03 := "BK02"."X13-1.TAPE TOP DOWN",
                     signal04 := "BK02"."X14-1.TAPE BTM DOWN",
                     signal05 := "BK02"."X15-1.SPLICE HEAD ROTATE TOP BACKWARD",
                     signal06 := "BK02"."X16-1.SPLICE HEAD ROTATE BTM BACKWARD",
                     signal07 := "BK02"."X17-1.SPARE",
                     signal08 := "BK02"."X10-2.SUCTION PAD TOP UP",
                     signal09 := "BK02"."X11-2.SUCTION PAD BTM UP",
                     signal10 := "BK02"."X12-2.CUTTER UP",
                     signal11 := "BK02"."X13-2.TAPE TOP UP",
                     signal12 := "BK02"."X14-2.TAPE BTM UP",
                     signal13 := "BK02"."X15-2.SPLICE HEAD ROTATE TOP FORWARD",
                     signal14 := "BK02"."X16-2.SPLICE HEAD ROTATE BTM FORWARD",
                     signal15 := "BK02"."X17-2.SPARE",
                     interfaceSignals := #statInterfaceSignalsHmi[5].valueSymbolLeft,
                     ENO => #_w1);
   IF #_w1 THEN
       #instSignals5Right(interfaceSignals := #statInterfaceSignalsHmi[5].valueSymbolRight);   // "LAF_InterfaceSignalsBool"
   END_IF;
END_REGION

REGION Network 11: Interface Signals 05 -Example: Model Flex-Pro-Line - IN/OUT- / Interface Signals 06
   // Aufruf des Schnittstellen Signal Bausteins Ba-Bereich 4 / Call the interface signals bool blocks of opmode 4
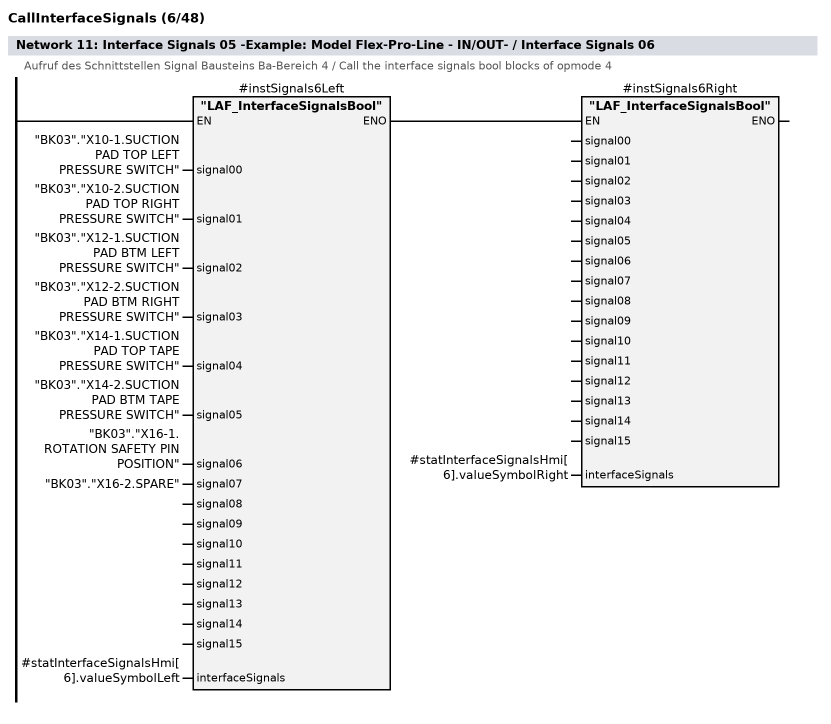
   RUNG wire#powerrail
      #instSignals6Left(signal00 := "BK03"."X10-1.SUCTION PAD TOP LEFT PRESSURE SWITCH", signal01 := "BK03"."X10-2.SUCTION PAD TOP RIGHT PRESSURE SWITCH", signal02 := "BK03"."X12-1.SUCTION PAD BTM LEFT PRESSURE SWITCH", signal03 := "BK03"."X12-2.SUCTION PAD BTM RIGHT PRESSURE SWITCH", signal04 := "BK03"."X14-1.SUCTION PAD TOP TAPE PRESSURE SWITCH", signal05 := "BK03"."X14-2.SUCTION PAD BTM TAPE PRESSURE SWITCH", signal06 := "BK03"."X16-1.ROTATION SAFETY PIN POSITION", signal07 := "BK03"."X16-2.SPARE", signal08 :=, signal09 :=, signal10 :=, signal11 :=, signal12 :=, signal13 :=, signal14 :=, signal15 :=, interfaceSignals := #statInterfaceSignalsHmi[6].valueSymbolLeft)
      #instSignals6Right(signal00 :=, signal01 :=, signal02 :=, signal03 :=, signal04 :=, signal05 :=, signal06 :=, signal07 :=, signal08 :=, signal09 :=, signal10 :=, signal11 :=, signal12 :=, signal13 :=, signal14 :=, signal15 :=, interfaceSignals := #statInterfaceSignalsHmi[6].valueSymbolRight)
   END_RUNG
   // the same network as SCL:
   #instSignals6Left(signal00 := "BK03"."X10-1.SUCTION PAD TOP LEFT PRESSURE SWITCH",   // "LAF_InterfaceSignalsBool"
                     signal01 := "BK03"."X10-2.SUCTION PAD TOP RIGHT PRESSURE SWITCH",
                     signal02 := "BK03"."X12-1.SUCTION PAD BTM LEFT PRESSURE SWITCH",
                     signal03 := "BK03"."X12-2.SUCTION PAD BTM RIGHT PRESSURE SWITCH",
                     signal04 := "BK03"."X14-1.SUCTION PAD TOP TAPE PRESSURE SWITCH",
                     signal05 := "BK03"."X14-2.SUCTION PAD BTM TAPE PRESSURE SWITCH",
                     signal06 := "BK03"."X16-1.ROTATION SAFETY PIN POSITION",
                     signal07 := "BK03"."X16-2.SPARE",
                     interfaceSignals := #statInterfaceSignalsHmi[6].valueSymbolLeft,
                     ENO => #_w1);
   IF #_w1 THEN
       #instSignals6Right(interfaceSignals := #statInterfaceSignalsHmi[6].valueSymbolRight);   // "LAF_InterfaceSignalsBool"
   END_IF;
END_REGION

REGION Network 12: Interface Signals 05 -Example: Model Flex-Pro-Line - IN/OUT- / Interface Signals 07
   // Aufruf des Schnittstellen Signal Bausteins Ba-Bereich 4 / Call the interface signals bool blocks of opmode 4
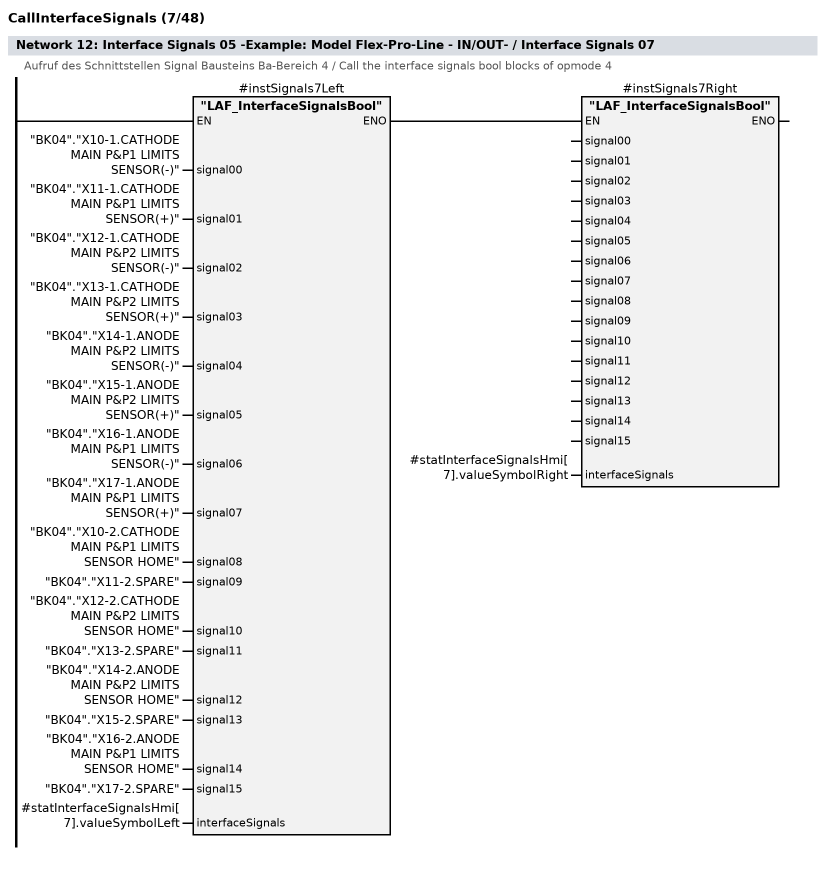
   RUNG wire#powerrail
      #instSignals7Left(signal00 := "BK04"."X10-1.CATHODE MAIN P&P1 LIMITS SENSOR(-)", signal01 := "BK04"."X11-1.CATHODE MAIN P&P1 LIMITS SENSOR(+)", signal02 := "BK04"."X12-1.CATHODE MAIN P&P2 LIMITS SENSOR(-)", signal03 := "BK04"."X13-1.CATHODE MAIN P&P2 LIMITS SENSOR(+)", signal04 := "BK04"."X14-1.ANODE MAIN P&P2 LIMITS SENSOR(-)", signal05 := "BK04"."X15-1.ANODE MAIN P&P2 LIMITS SENSOR(+)", signal06 := "BK04"."X16-1.ANODE MAIN P&P1 LIMITS SENSOR(-)", signal07 := "BK04"."X17-1.ANODE MAIN P&P1 LIMITS SENSOR(+)", signal08 := "BK04"."X10-2.CATHODE MAIN P&P1 LIMITS SENSOR HOME", signal09 := "BK04"."X11-2.SPARE", signal10 := "BK04"."X12-2.CATHODE MAIN P&P2 LIMITS SENSOR HOME", signal11 := "BK04"."X13-2.SPARE", signal12 := "BK04"."X14-2.ANODE MAIN P&P2 LIMITS SENSOR HOME", signal13 := "BK04"."X15-2.SPARE", signal14 := "BK04"."X16-2.ANODE MAIN P&P1 LIMITS SENSOR HOME", signal15 := "BK04"."X17-2.SPARE", interfaceSignals := #statInterfaceSignalsHmi[7].valueSymbolLeft)
      #instSignals7Right(signal00 :=, signal01 :=, signal02 :=, signal03 :=, signal04 :=, signal05 :=, signal06 :=, signal07 :=, signal08 :=, signal09 :=, signal10 :=, signal11 :=, signal12 :=, signal13 :=, signal14 :=, signal15 :=, interfaceSignals := #statInterfaceSignalsHmi[7].valueSymbolRight)
   END_RUNG
   // the same network as SCL:
   #instSignals7Left(signal00 := "BK04"."X10-1.CATHODE MAIN P&P1 LIMITS SENSOR(-)",   // "LAF_InterfaceSignalsBool"
                     signal01 := "BK04"."X11-1.CATHODE MAIN P&P1 LIMITS SENSOR(+)",
                     signal02 := "BK04"."X12-1.CATHODE MAIN P&P2 LIMITS SENSOR(-)",
                     signal03 := "BK04"."X13-1.CATHODE MAIN P&P2 LIMITS SENSOR(+)",
                     signal04 := "BK04"."X14-1.ANODE MAIN P&P2 LIMITS SENSOR(-)",
                     signal05 := "BK04"."X15-1.ANODE MAIN P&P2 LIMITS SENSOR(+)",
                     signal06 := "BK04"."X16-1.ANODE MAIN P&P1 LIMITS SENSOR(-)",
                     signal07 := "BK04"."X17-1.ANODE MAIN P&P1 LIMITS SENSOR(+)",
                     signal08 := "BK04"."X10-2.CATHODE MAIN P&P1 LIMITS SENSOR HOME",
                     signal09 := "BK04"."X11-2.SPARE",
                     signal10 := "BK04"."X12-2.CATHODE MAIN P&P2 LIMITS SENSOR HOME",
                     signal11 := "BK04"."X13-2.SPARE",
                     signal12 := "BK04"."X14-2.ANODE MAIN P&P2 LIMITS SENSOR HOME",
                     signal13 := "BK04"."X15-2.SPARE",
                     signal14 := "BK04"."X16-2.ANODE MAIN P&P1 LIMITS SENSOR HOME",
                     signal15 := "BK04"."X17-2.SPARE",
                     interfaceSignals := #statInterfaceSignalsHmi[7].valueSymbolLeft,
                     ENO => #_w1);
   IF #_w1 THEN
       #instSignals7Right(interfaceSignals := #statInterfaceSignalsHmi[7].valueSymbolRight);   // "LAF_InterfaceSignalsBool"
   END_IF;
END_REGION

REGION Network 13: Interface Signals 05 -Example: Model Flex-Pro-Line - IN/OUT- / Interface Signals 08
   // Aufruf des Schnittstellen Signal Bausteins Ba-Bereich 4 / Call the interface signals bool blocks of opmode 4
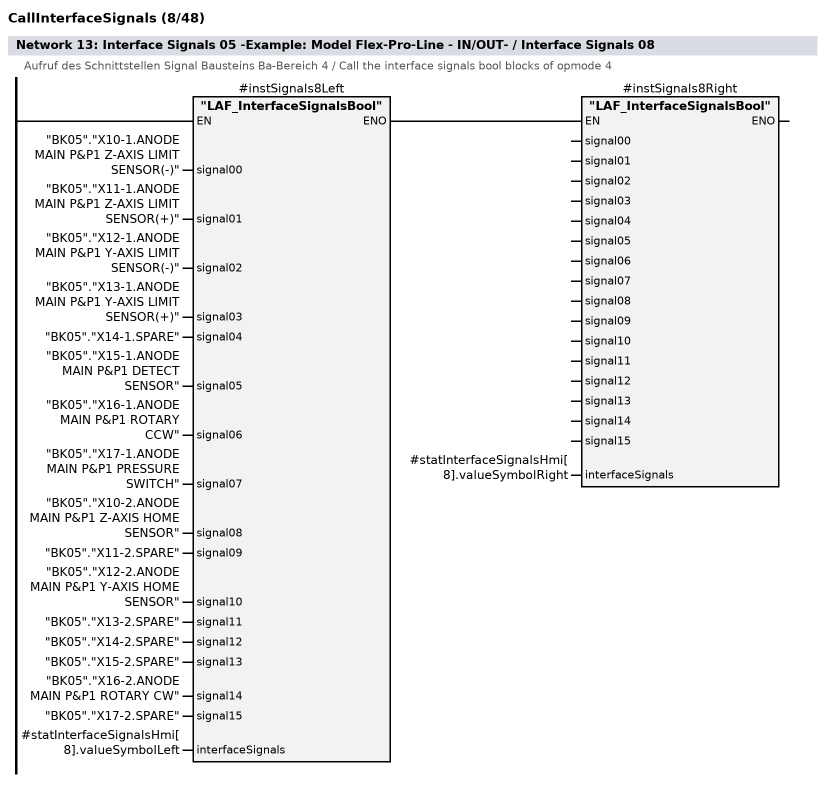
   RUNG wire#powerrail
      #instSignals8Left(signal00 := "BK05"."X10-1.ANODE MAIN P&P1 Z-AXIS LIMIT SENSOR(-)", signal01 := "BK05"."X11-1.ANODE MAIN P&P1 Z-AXIS LIMIT SENSOR(+)", signal02 := "BK05"."X12-1.ANODE MAIN P&P1 Y-AXIS LIMIT SENSOR(-)", signal03 := "BK05"."X13-1.ANODE MAIN P&P1 Y-AXIS LIMIT SENSOR(+)", signal04 := "BK05"."X14-1.SPARE", signal05 := "BK05"."X15-1.ANODE MAIN P&P1 DETECT SENSOR", signal06 := "BK05"."X16-1.ANODE MAIN P&P1 ROTARY CCW", signal07 := "BK05"."X17-1.ANODE MAIN P&P1 PRESSURE SWITCH", signal08 := "BK05"."X10-2.ANODE MAIN P&P1 Z-AXIS HOME SENSOR", signal09 := "BK05"."X11-2.SPARE", signal10 := "BK05"."X12-2.ANODE MAIN P&P1 Y-AXIS HOME SENSOR", signal11 := "BK05"."X13-2.SPARE", signal12 := "BK05"."X14-2.SPARE", signal13 := "BK05"."X15-2.SPARE", signal14 := "BK05"."X16-2.ANODE MAIN P&P1 ROTARY CW", signal15 := "BK05"."X17-2.SPARE", interfaceSignals := #statInterfaceSignalsHmi[8].valueSymbolLeft)
      #instSignals8Right(signal00 :=, signal01 :=, signal02 :=, signal03 :=, signal04 :=, signal05 :=, signal06 :=, signal07 :=, signal08 :=, signal09 :=, signal10 :=, signal11 :=, signal12 :=, signal13 :=, signal14 :=, signal15 :=, interfaceSignals := #statInterfaceSignalsHmi[8].valueSymbolRight)
   END_RUNG
   // the same network as SCL:
   #instSignals8Left(signal00 := "BK05"."X10-1.ANODE MAIN P&P1 Z-AXIS LIMIT SENSOR(-)",   // "LAF_InterfaceSignalsBool"
                     signal01 := "BK05"."X11-1.ANODE MAIN P&P1 Z-AXIS LIMIT SENSOR(+)",
                     signal02 := "BK05"."X12-1.ANODE MAIN P&P1 Y-AXIS LIMIT SENSOR(-)",
                     signal03 := "BK05"."X13-1.ANODE MAIN P&P1 Y-AXIS LIMIT SENSOR(+)",
                     signal04 := "BK05"."X14-1.SPARE",
                     signal05 := "BK05"."X15-1.ANODE MAIN P&P1 DETECT SENSOR",
                     signal06 := "BK05"."X16-1.ANODE MAIN P&P1 ROTARY CCW",
                     signal07 := "BK05"."X17-1.ANODE MAIN P&P1 PRESSURE SWITCH",
                     signal08 := "BK05"."X10-2.ANODE MAIN P&P1 Z-AXIS HOME SENSOR",
                     signal09 := "BK05"."X11-2.SPARE",
                     signal10 := "BK05"."X12-2.ANODE MAIN P&P1 Y-AXIS HOME SENSOR",
                     signal11 := "BK05"."X13-2.SPARE",
                     signal12 := "BK05"."X14-2.SPARE",
                     signal13 := "BK05"."X15-2.SPARE",
                     signal14 := "BK05"."X16-2.ANODE MAIN P&P1 ROTARY CW",
                     signal15 := "BK05"."X17-2.SPARE",
                     interfaceSignals := #statInterfaceSignalsHmi[8].valueSymbolLeft,
                     ENO => #_w1);
   IF #_w1 THEN
       #instSignals8Right(interfaceSignals := #statInterfaceSignalsHmi[8].valueSymbolRight);   // "LAF_InterfaceSignalsBool"
   END_IF;
END_REGION

REGION Network 14: Interface Signals 05 -Example: Model Flex-Pro-Line - IN/OUT- / Interface Signals 09
   // Aufruf des Schnittstellen Signal Bausteins Ba-Bereich 4 / Call the interface signals bool blocks of opmode 4
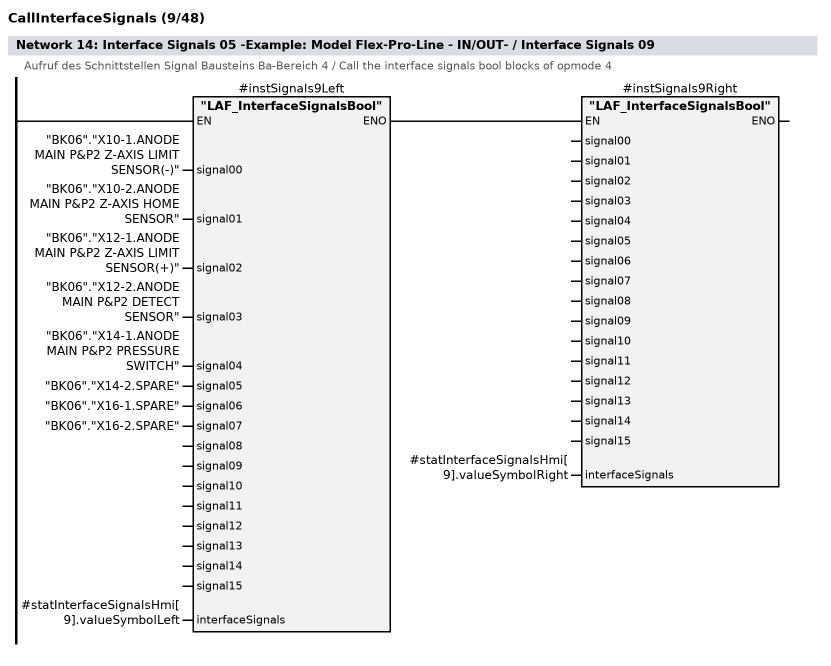
   RUNG wire#powerrail
      #instSignals9Left(signal00 := "BK06"."X10-1.ANODE MAIN P&P2 Z-AXIS LIMIT SENSOR(-)", signal01 := "BK06"."X10-2.ANODE MAIN P&P2 Z-AXIS HOME SENSOR", signal02 := "BK06"."X12-1.ANODE MAIN P&P2 Z-AXIS LIMIT SENSOR(+)", signal03 := "BK06"."X12-2.ANODE MAIN P&P2 DETECT SENSOR", signal04 := "BK06"."X14-1.ANODE MAIN P&P2 PRESSURE SWITCH", signal05 := "BK06"."X14-2.SPARE", signal06 := "BK06"."X16-1.SPARE", signal07 := "BK06"."X16-2.SPARE", signal08 :=, signal09 :=, signal10 :=, signal11 :=, signal12 :=, signal13 :=, signal14 :=, signal15 :=, interfaceSignals := #statInterfaceSignalsHmi[9].valueSymbolLeft)
      #instSignals9Right(signal00 :=, signal01 :=, signal02 :=, signal03 :=, signal04 :=, signal05 :=, signal06 :=, signal07 :=, signal08 :=, signal09 :=, signal10 :=, signal11 :=, signal12 :=, signal13 :=, signal14 :=, signal15 :=, interfaceSignals := #statInterfaceSignalsHmi[9].valueSymbolRight)
   END_RUNG
   // the same network as SCL:
   #instSignals9Left(signal00 := "BK06"."X10-1.ANODE MAIN P&P2 Z-AXIS LIMIT SENSOR(-)",   // "LAF_InterfaceSignalsBool"
                     signal01 := "BK06"."X10-2.ANODE MAIN P&P2 Z-AXIS HOME SENSOR",
                     signal02 := "BK06"."X12-1.ANODE MAIN P&P2 Z-AXIS LIMIT SENSOR(+)",
                     signal03 := "BK06"."X12-2.ANODE MAIN P&P2 DETECT SENSOR",
                     signal04 := "BK06"."X14-1.ANODE MAIN P&P2 PRESSURE SWITCH",
                     signal05 := "BK06"."X14-2.SPARE",
                     signal06 := "BK06"."X16-1.SPARE",
                     signal07 := "BK06"."X16-2.SPARE",
                     interfaceSignals := #statInterfaceSignalsHmi[9].valueSymbolLeft,
                     ENO => #_w1);
   IF #_w1 THEN
       #instSignals9Right(interfaceSignals := #statInterfaceSignalsHmi[9].valueSymbolRight);   // "LAF_InterfaceSignalsBool"
   END_IF;
END_REGION

REGION Network 15: Interface Signals 05 -Example: Model Flex-Pro-Line - IN/OUT- / Interface Signals 10
   // Aufruf des Schnittstellen Signal Bausteins Ba-Bereich 4 / Call the interface signals bool blocks of opmode 4
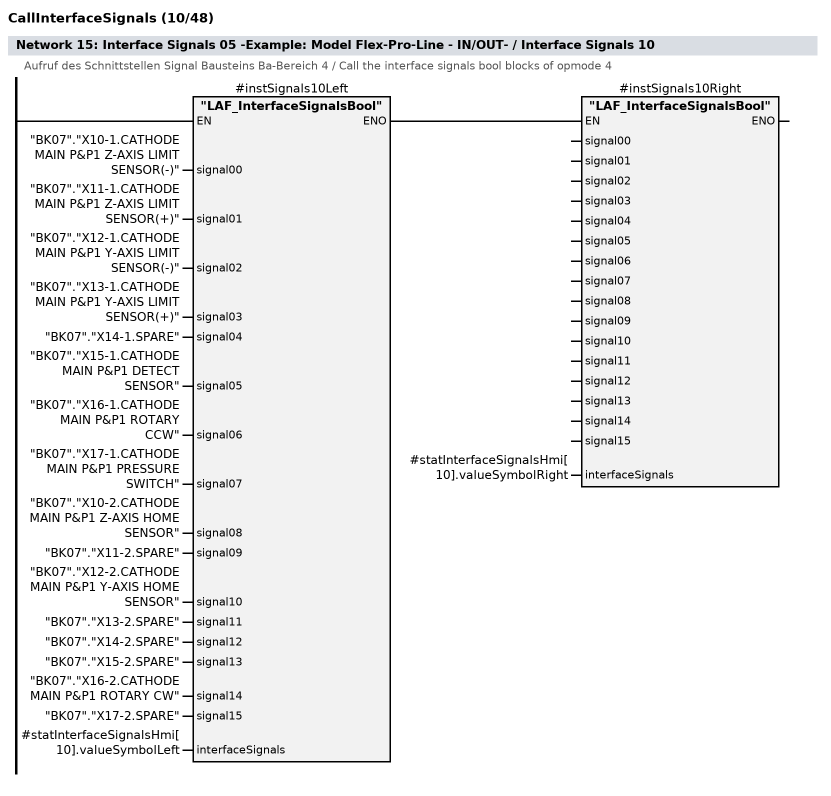
   RUNG wire#powerrail
      #instSignals10Left(signal00 := "BK07"."X10-1.CATHODE MAIN P&P1 Z-AXIS LIMIT SENSOR(-)", signal01 := "BK07"."X11-1.CATHODE MAIN P&P1 Z-AXIS LIMIT SENSOR(+)", signal02 := "BK07"."X12-1.CATHODE MAIN P&P1 Y-AXIS LIMIT SENSOR(-)", signal03 := "BK07"."X13-1.CATHODE MAIN P&P1 Y-AXIS LIMIT SENSOR(+)", signal04 := "BK07"."X14-1.SPARE", signal05 := "BK07"."X15-1.CATHODE MAIN P&P1 DETECT SENSOR", signal06 := "BK07"."X16-1.CATHODE MAIN P&P1 ROTARY CCW", signal07 := "BK07"."X17-1.CATHODE MAIN P&P1 PRESSURE SWITCH", signal08 := "BK07"."X10-2.CATHODE MAIN P&P1 Z-AXIS HOME SENSOR", signal09 := "BK07"."X11-2.SPARE", signal10 := "BK07"."X12-2.CATHODE MAIN P&P1 Y-AXIS HOME SENSOR", signal11 := "BK07"."X13-2.SPARE", signal12 := "BK07"."X14-2.SPARE", signal13 := "BK07"."X15-2.SPARE", signal14 := "BK07"."X16-2.CATHODE MAIN P&P1 ROTARY CW", signal15 := "BK07"."X17-2.SPARE", interfaceSignals := #statInterfaceSignalsHmi[10].valueSymbolLeft)
      #instSignals10Right(signal00 :=, signal01 :=, signal02 :=, signal03 :=, signal04 :=, signal05 :=, signal06 :=, signal07 :=, signal08 :=, signal09 :=, signal10 :=, signal11 :=, signal12 :=, signal13 :=, signal14 :=, signal15 :=, interfaceSignals := #statInterfaceSignalsHmi[10].valueSymbolRight)
   END_RUNG
   // the same network as SCL:
   #instSignals10Left(signal00 := "BK07"."X10-1.CATHODE MAIN P&P1 Z-AXIS LIMIT SENSOR(-)",   // "LAF_InterfaceSignalsBool"
                      signal01 := "BK07"."X11-1.CATHODE MAIN P&P1 Z-AXIS LIMIT SENSOR(+)",
                      signal02 := "BK07"."X12-1.CATHODE MAIN P&P1 Y-AXIS LIMIT SENSOR(-)",
                      signal03 := "BK07"."X13-1.CATHODE MAIN P&P1 Y-AXIS LIMIT SENSOR(+)",
                      signal04 := "BK07"."X14-1.SPARE",
                      signal05 := "BK07"."X15-1.CATHODE MAIN P&P1 DETECT SENSOR",
                      signal06 := "BK07"."X16-1.CATHODE MAIN P&P1 ROTARY CCW",
                      signal07 := "BK07"."X17-1.CATHODE MAIN P&P1 PRESSURE SWITCH",
                      signal08 := "BK07"."X10-2.CATHODE MAIN P&P1 Z-AXIS HOME SENSOR",
                      signal09 := "BK07"."X11-2.SPARE",
                      signal10 := "BK07"."X12-2.CATHODE MAIN P&P1 Y-AXIS HOME SENSOR",
                      signal11 := "BK07"."X13-2.SPARE",
                      signal12 := "BK07"."X14-2.SPARE",
                      signal13 := "BK07"."X15-2.SPARE",
                      signal14 := "BK07"."X16-2.CATHODE MAIN P&P1 ROTARY CW",
                      signal15 := "BK07"."X17-2.SPARE",
                      interfaceSignals := #statInterfaceSignalsHmi[10].valueSymbolLeft,
                      ENO => #_w1);
   IF #_w1 THEN
       #instSignals10Right(interfaceSignals := #statInterfaceSignalsHmi[10].valueSymbolRight);   // "LAF_InterfaceSignalsBool"
   END_IF;
END_REGION

REGION Network 16: Interface Signals 05 -Example: Model Flex-Pro-Line - IN/OUT- / Interface Signals 11
   // Aufruf des Schnittstellen Signal Bausteins Ba-Bereich 4 / Call the interface signals bool blocks of opmode 4
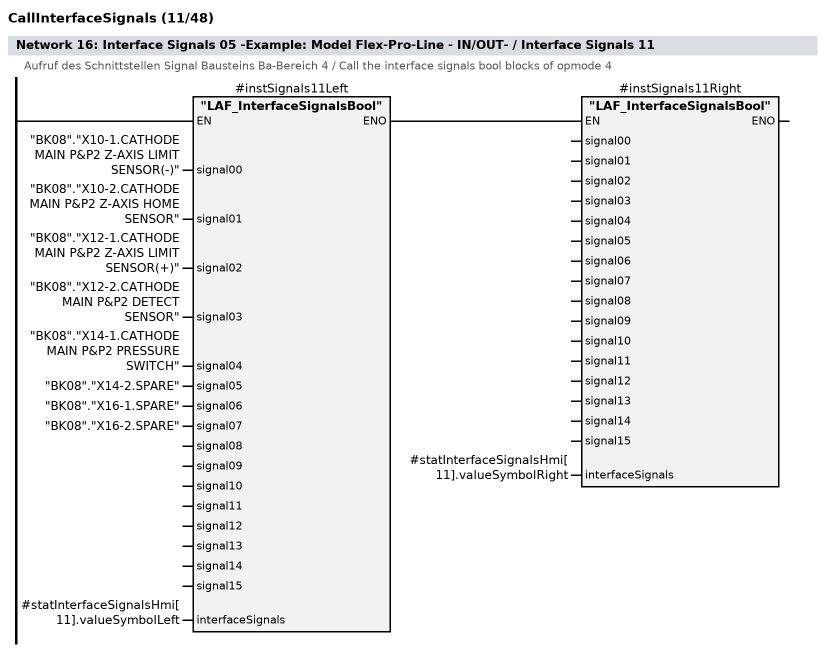
   RUNG wire#powerrail
      #instSignals11Left(signal00 := "BK08"."X10-1.CATHODE MAIN P&P2 Z-AXIS LIMIT SENSOR(-)", signal01 := "BK08"."X10-2.CATHODE MAIN P&P2 Z-AXIS HOME SENSOR", signal02 := "BK08"."X12-1.CATHODE MAIN P&P2 Z-AXIS LIMIT SENSOR(+)", signal03 := "BK08"."X12-2.CATHODE MAIN P&P2 DETECT SENSOR", signal04 := "BK08"."X14-1.CATHODE MAIN P&P2 PRESSURE SWITCH", signal05 := "BK08"."X14-2.SPARE", signal06 := "BK08"."X16-1.SPARE", signal07 := "BK08"."X16-2.SPARE", signal08 :=, signal09 :=, signal10 :=, signal11 :=, signal12 :=, signal13 :=, signal14 :=, signal15 :=, interfaceSignals := #statInterfaceSignalsHmi[11].valueSymbolLeft)
      #instSignals11Right(signal00 :=, signal01 :=, signal02 :=, signal03 :=, signal04 :=, signal05 :=, signal06 :=, signal07 :=, signal08 :=, signal09 :=, signal10 :=, signal11 :=, signal12 :=, signal13 :=, signal14 :=, signal15 :=, interfaceSignals := #statInterfaceSignalsHmi[11].valueSymbolRight)
   END_RUNG
   // the same network as SCL:
   #instSignals11Left(signal00 := "BK08"."X10-1.CATHODE MAIN P&P2 Z-AXIS LIMIT SENSOR(-)",   // "LAF_InterfaceSignalsBool"
                      signal01 := "BK08"."X10-2.CATHODE MAIN P&P2 Z-AXIS HOME SENSOR",
                      signal02 := "BK08"."X12-1.CATHODE MAIN P&P2 Z-AXIS LIMIT SENSOR(+)",
                      signal03 := "BK08"."X12-2.CATHODE MAIN P&P2 DETECT SENSOR",
                      signal04 := "BK08"."X14-1.CATHODE MAIN P&P2 PRESSURE SWITCH",
                      signal05 := "BK08"."X14-2.SPARE",
                      signal06 := "BK08"."X16-1.SPARE",
                      signal07 := "BK08"."X16-2.SPARE",
                      interfaceSignals := #statInterfaceSignalsHmi[11].valueSymbolLeft,
                      ENO => #_w1);
   IF #_w1 THEN
       #instSignals11Right(interfaceSignals := #statInterfaceSignalsHmi[11].valueSymbolRight);   // "LAF_InterfaceSignalsBool"
   END_IF;
END_REGION

REGION Network 17: Interface Signals 05 -Example: Model Flex-Pro-Line - IN/OUT- / Interface Signals 12
   // Aufruf des Schnittstellen Signal Bausteins Ba-Bereich 4 / Call the interface signals bool blocks of opmode 4
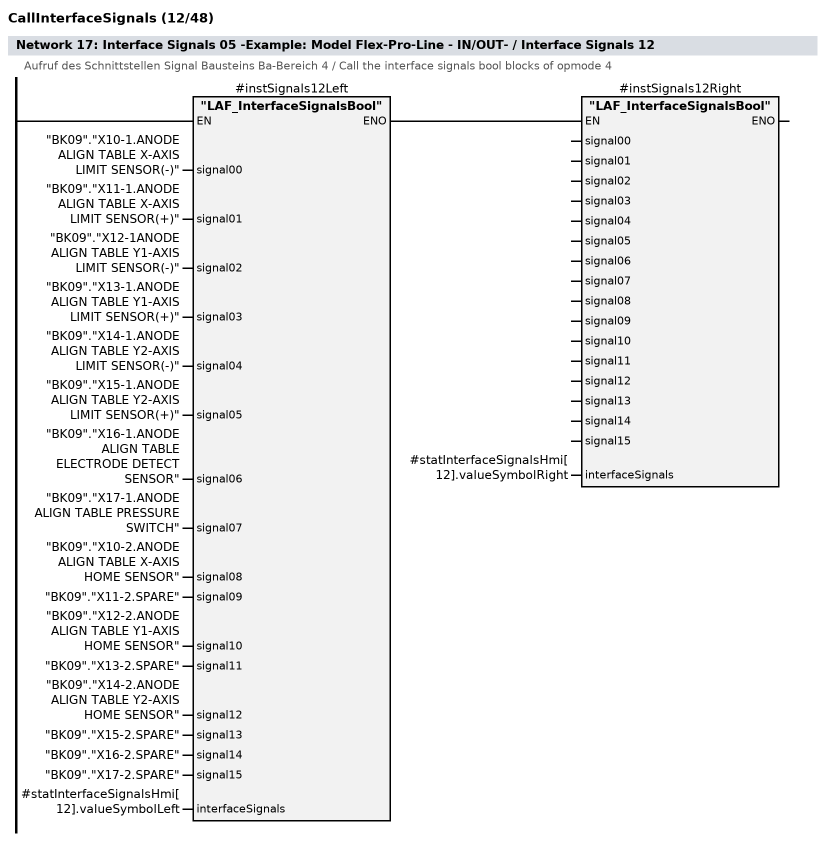
   RUNG wire#powerrail
      #instSignals12Left(signal00 := "BK09"."X10-1.ANODE ALIGN TABLE X-AXIS LIMIT SENSOR(-)", signal01 := "BK09"."X11-1.ANODE ALIGN TABLE X-AXIS LIMIT SENSOR(+)", signal02 := "BK09"."X12-1ANODE ALIGN TABLE Y1-AXIS LIMIT SENSOR(-)", signal03 := "BK09"."X13-1.ANODE ALIGN TABLE Y1-AXIS LIMIT SENSOR(+)", signal04 := "BK09"."X14-1.ANODE ALIGN TABLE Y2-AXIS LIMIT SENSOR(-)", signal05 := "BK09"."X15-1.ANODE ALIGN TABLE Y2-AXIS LIMIT SENSOR(+)", signal06 := "BK09"."X16-1.ANODE ALIGN TABLE ELECTRODE DETECT SENSOR", signal07 := "BK09"."X17-1.ANODE ALIGN TABLE PRESSURE SWITCH", signal08 := "BK09"."X10-2.ANODE ALIGN TABLE X-AXIS HOME SENSOR", signal09 := "BK09"."X11-2.SPARE", signal10 := "BK09"."X12-2.ANODE ALIGN TABLE Y1-AXIS HOME SENSOR", signal11 := "BK09"."X13-2.SPARE", signal12 := "BK09"."X14-2.ANODE ALIGN TABLE Y2-AXIS HOME SENSOR", signal13 := "BK09"."X15-2.SPARE", signal14 := "BK09"."X16-2.SPARE", signal15 := "BK09"."X17-2.SPARE", interfaceSignals := #statInterfaceSignalsHmi[12].valueSymbolLeft)
      #instSignals12Right(signal00 :=, signal01 :=, signal02 :=, signal03 :=, signal04 :=, signal05 :=, signal06 :=, signal07 :=, signal08 :=, signal09 :=, signal10 :=, signal11 :=, signal12 :=, signal13 :=, signal14 :=, signal15 :=, interfaceSignals := #statInterfaceSignalsHmi[12].valueSymbolRight)
   END_RUNG
   // the same network as SCL:
   #instSignals12Left(signal00 := "BK09"."X10-1.ANODE ALIGN TABLE X-AXIS LIMIT SENSOR(-)",   // "LAF_InterfaceSignalsBool"
                      signal01 := "BK09"."X11-1.ANODE ALIGN TABLE X-AXIS LIMIT SENSOR(+)",
                      signal02 := "BK09"."X12-1ANODE ALIGN TABLE Y1-AXIS LIMIT SENSOR(-)",
                      signal03 := "BK09"."X13-1.ANODE ALIGN TABLE Y1-AXIS LIMIT SENSOR(+)",
                      signal04 := "BK09"."X14-1.ANODE ALIGN TABLE Y2-AXIS LIMIT SENSOR(-)",
                      signal05 := "BK09"."X15-1.ANODE ALIGN TABLE Y2-AXIS LIMIT SENSOR(+)",
                      signal06 := "BK09"."X16-1.ANODE ALIGN TABLE ELECTRODE DETECT SENSOR",
                      signal07 := "BK09"."X17-1.ANODE ALIGN TABLE PRESSURE SWITCH",
                      signal08 := "BK09"."X10-2.ANODE ALIGN TABLE X-AXIS HOME SENSOR",
                      signal09 := "BK09"."X11-2.SPARE",
                      signal10 := "BK09"."X12-2.ANODE ALIGN TABLE Y1-AXIS HOME SENSOR",
                      signal11 := "BK09"."X13-2.SPARE",
                      signal12 := "BK09"."X14-2.ANODE ALIGN TABLE Y2-AXIS HOME SENSOR",
                      signal13 := "BK09"."X15-2.SPARE",
                      signal14 := "BK09"."X16-2.SPARE",
                      signal15 := "BK09"."X17-2.SPARE",
                      interfaceSignals := #statInterfaceSignalsHmi[12].valueSymbolLeft,
                      ENO => #_w1);
   IF #_w1 THEN
       #instSignals12Right(interfaceSignals := #statInterfaceSignalsHmi[12].valueSymbolRight);   // "LAF_InterfaceSignalsBool"
   END_IF;
END_REGION

REGION Network 18: Interface Signals 03 -Example: System flags & Clock flags- / Interface Signals13
   // Aufruf des Schnittstellen Signal Bausteins für die Systemvariablen / Call the interface signals bool blocks of system tags
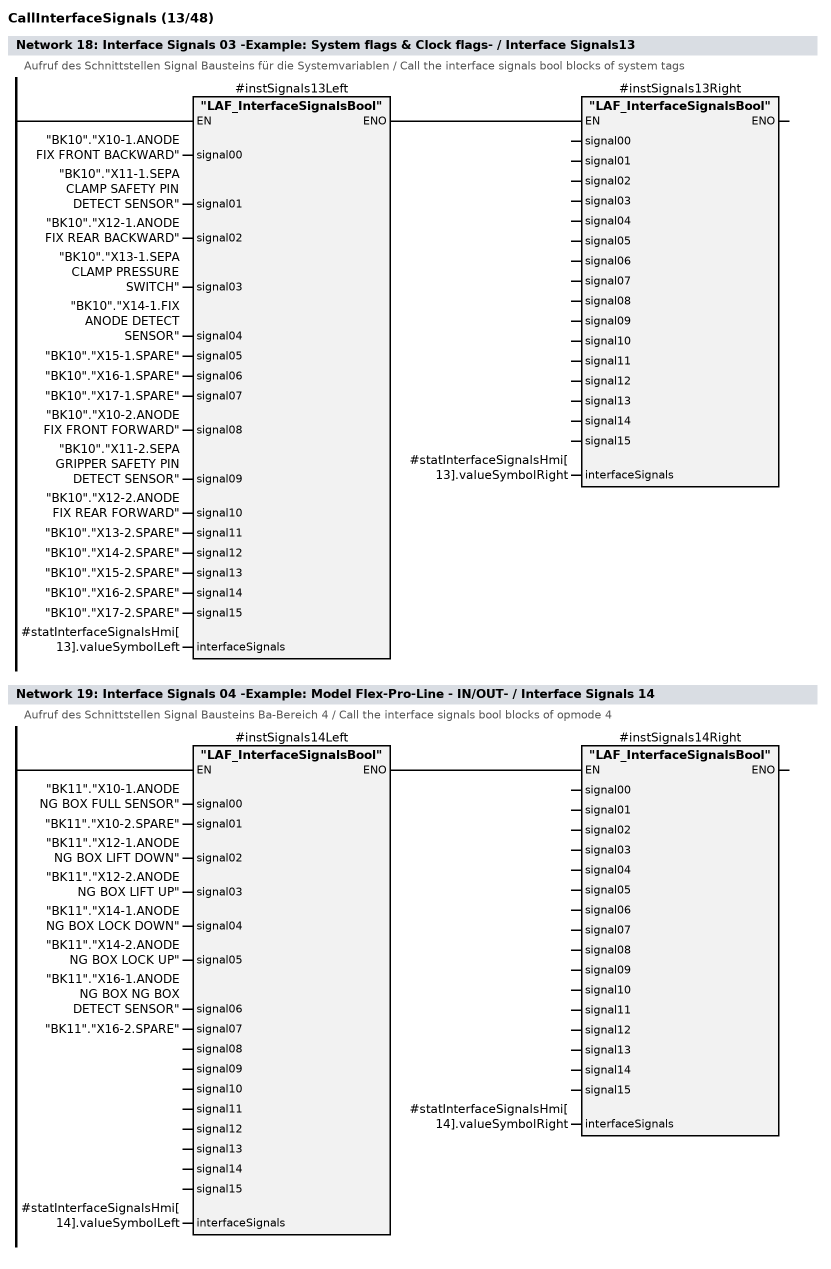
   RUNG wire#powerrail
      #instSignals13Left(signal00 := "BK10"."X10-1.ANODE FIX FRONT BACKWARD", signal01 := "BK10"."X11-1.SEPA CLAMP SAFETY PIN DETECT SENSOR", signal02 := "BK10"."X12-1.ANODE FIX REAR BACKWARD", signal03 := "BK10"."X13-1.SEPA CLAMP PRESSURE SWITCH", signal04 := "BK10"."X14-1.FIX ANODE DETECT SENSOR", signal05 := "BK10"."X15-1.SPARE", signal06 := "BK10"."X16-1.SPARE", signal07 := "BK10"."X17-1.SPARE", signal08 := "BK10"."X10-2.ANODE FIX FRONT FORWARD", signal09 := "BK10"."X11-2.SEPA GRIPPER SAFETY PIN DETECT SENSOR", signal10 := "BK10"."X12-2.ANODE FIX REAR FORWARD", signal11 := "BK10"."X13-2.SPARE", signal12 := "BK10"."X14-2.SPARE", signal13 := "BK10"."X15-2.SPARE", signal14 := "BK10"."X16-2.SPARE", signal15 := "BK10"."X17-2.SPARE", interfaceSignals := #statInterfaceSignalsHmi[13].valueSymbolLeft)
      #instSignals13Right(signal00 :=, signal01 :=, signal02 :=, signal03 :=, signal04 :=, signal05 :=, signal06 :=, signal07 :=, signal08 :=, signal09 :=, signal10 :=, signal11 :=, signal12 :=, signal13 :=, signal14 :=, signal15 :=, interfaceSignals := #statInterfaceSignalsHmi[13].valueSymbolRight)
   END_RUNG
   // the same network as SCL:
   #instSignals13Left(signal00 := "BK10"."X10-1.ANODE FIX FRONT BACKWARD",   // "LAF_InterfaceSignalsBool"
                      signal01 := "BK10"."X11-1.SEPA CLAMP SAFETY PIN DETECT SENSOR",
                      signal02 := "BK10"."X12-1.ANODE FIX REAR BACKWARD",
                      signal03 := "BK10"."X13-1.SEPA CLAMP PRESSURE SWITCH",
                      signal04 := "BK10"."X14-1.FIX ANODE DETECT SENSOR",
                      signal05 := "BK10"."X15-1.SPARE",
                      signal06 := "BK10"."X16-1.SPARE",
                      signal07 := "BK10"."X17-1.SPARE",
                      signal08 := "BK10"."X10-2.ANODE FIX FRONT FORWARD",
                      signal09 := "BK10"."X11-2.SEPA GRIPPER SAFETY PIN DETECT SENSOR",
                      signal10 := "BK10"."X12-2.ANODE FIX REAR FORWARD",
                      signal11 := "BK10"."X13-2.SPARE",
                      signal12 := "BK10"."X14-2.SPARE",
                      signal13 := "BK10"."X15-2.SPARE",
                      signal14 := "BK10"."X16-2.SPARE",
                      signal15 := "BK10"."X17-2.SPARE",
                      interfaceSignals := #statInterfaceSignalsHmi[13].valueSymbolLeft,
                      ENO => #_w1);
   IF #_w1 THEN
       #instSignals13Right(interfaceSignals := #statInterfaceSignalsHmi[13].valueSymbolRight);   // "LAF_InterfaceSignalsBool"
   END_IF;
END_REGION

REGION Network 19: Interface Signals 04 -Example: Model Flex-Pro-Line - IN/OUT- / Interface Signals 14
   // Aufruf des Schnittstellen Signal Bausteins Ba-Bereich 4 / Call the interface signals bool blocks of opmode 4
   RUNG wire#powerrail
      #instSignals14Left(signal00 := "BK11"."X10-1.ANODE NG BOX FULL SENSOR", signal01 := "BK11"."X10-2.SPARE", signal02 := "BK11"."X12-1.ANODE NG BOX LIFT DOWN", signal03 := "BK11"."X12-2.ANODE NG BOX LIFT UP", signal04 := "BK11"."X14-1.ANODE NG BOX LOCK DOWN", signal05 := "BK11"."X14-2.ANODE NG BOX LOCK UP", signal06 := "BK11"."X16-1.ANODE NG BOX NG BOX DETECT SENSOR", signal07 := "BK11"."X16-2.SPARE", signal08 :=, signal09 :=, signal10 :=, signal11 :=, signal12 :=, signal13 :=, signal14 :=, signal15 :=, interfaceSignals := #statInterfaceSignalsHmi[14].valueSymbolLeft)
      #instSignals14Right(signal00 :=, signal01 :=, signal02 :=, signal03 :=, signal04 :=, signal05 :=, signal06 :=, signal07 :=, signal08 :=, signal09 :=, signal10 :=, signal11 :=, signal12 :=, signal13 :=, signal14 :=, signal15 :=, interfaceSignals := #statInterfaceSignalsHmi[14].valueSymbolRight)
   END_RUNG
   // the same network as SCL:
   #instSignals14Left(signal00 := "BK11"."X10-1.ANODE NG BOX FULL SENSOR",   // "LAF_InterfaceSignalsBool"
                      signal01 := "BK11"."X10-2.SPARE",
                      signal02 := "BK11"."X12-1.ANODE NG BOX LIFT DOWN",
                      signal03 := "BK11"."X12-2.ANODE NG BOX LIFT UP",
                      signal04 := "BK11"."X14-1.ANODE NG BOX LOCK DOWN",
                      signal05 := "BK11"."X14-2.ANODE NG BOX LOCK UP",
                      signal06 := "BK11"."X16-1.ANODE NG BOX NG BOX DETECT SENSOR",
                      signal07 := "BK11"."X16-2.SPARE",
                      interfaceSignals := #statInterfaceSignalsHmi[14].valueSymbolLeft,
                      ENO => #_w1);
   IF #_w1 THEN
       #instSignals14Right(interfaceSignals := #statInterfaceSignalsHmi[14].valueSymbolRight);   // "LAF_InterfaceSignalsBool"
   END_IF;
END_REGION

REGION Network 20: Interface Signals 05 -Example: Model Flex-Pro-Line - IN/OUT- / Interface Signals 15
   // Aufruf des Schnittstellen Signal Bausteins Ba-Bereich 4 / Call the interface signals bool blocks of opmode 4
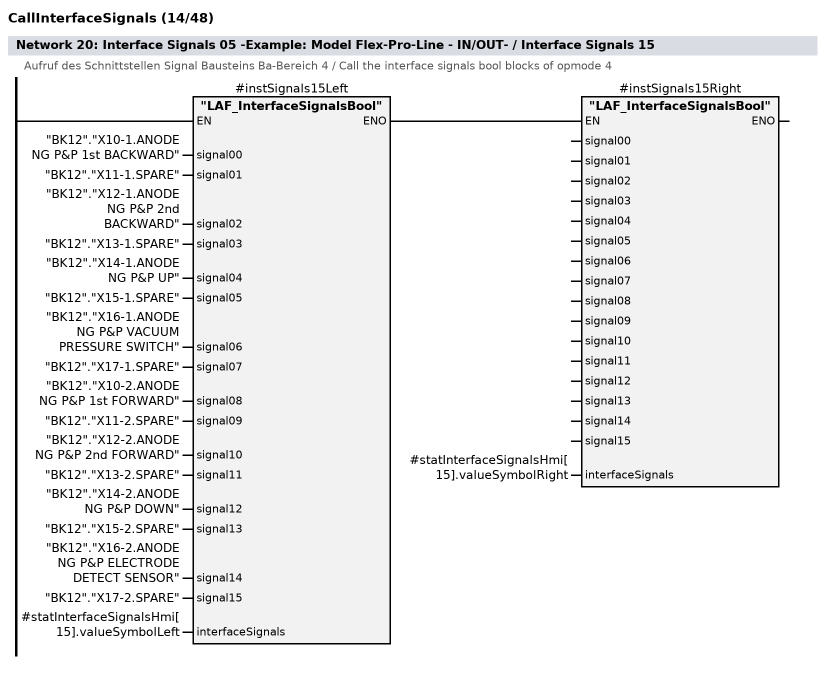
   RUNG wire#powerrail
      #instSignals15Left(signal00 := "BK12"."X10-1.ANODE NG P&P 1st BACKWARD", signal01 := "BK12"."X11-1.SPARE", signal02 := "BK12"."X12-1.ANODE NG P&P 2nd BACKWARD", signal03 := "BK12"."X13-1.SPARE", signal04 := "BK12"."X14-1.ANODE NG P&P UP", signal05 := "BK12"."X15-1.SPARE", signal06 := "BK12"."X16-1.ANODE NG P&P VACUUM PRESSURE SWITCH", signal07 := "BK12"."X17-1.SPARE", signal08 := "BK12"."X10-2.ANODE NG P&P 1st FORWARD", signal09 := "BK12"."X11-2.SPARE", signal10 := "BK12"."X12-2.ANODE NG P&P 2nd FORWARD", signal11 := "BK12"."X13-2.SPARE", signal12 := "BK12"."X14-2.ANODE NG P&P DOWN", signal13 := "BK12"."X15-2.SPARE", signal14 := "BK12"."X16-2.ANODE NG P&P ELECTRODE DETECT SENSOR", signal15 := "BK12"."X17-2.SPARE", interfaceSignals := #statInterfaceSignalsHmi[15].valueSymbolLeft)
      #instSignals15Right(signal00 :=, signal01 :=, signal02 :=, signal03 :=, signal04 :=, signal05 :=, signal06 :=, signal07 :=, signal08 :=, signal09 :=, signal10 :=, signal11 :=, signal12 :=, signal13 :=, signal14 :=, signal15 :=, interfaceSignals := #statInterfaceSignalsHmi[15].valueSymbolRight)
   END_RUNG
   // the same network as SCL:
   #instSignals15Left(signal00 := "BK12"."X10-1.ANODE NG P&P 1st BACKWARD",   // "LAF_InterfaceSignalsBool"
                      signal01 := "BK12"."X11-1.SPARE",
                      signal02 := "BK12"."X12-1.ANODE NG P&P 2nd BACKWARD",
                      signal03 := "BK12"."X13-1.SPARE",
                      signal04 := "BK12"."X14-1.ANODE NG P&P UP",
                      signal05 := "BK12"."X15-1.SPARE",
                      signal06 := "BK12"."X16-1.ANODE NG P&P VACUUM PRESSURE SWITCH",
                      signal07 := "BK12"."X17-1.SPARE",
                      signal08 := "BK12"."X10-2.ANODE NG P&P 1st FORWARD",
                      signal09 := "BK12"."X11-2.SPARE",
                      signal10 := "BK12"."X12-2.ANODE NG P&P 2nd FORWARD",
                      signal11 := "BK12"."X13-2.SPARE",
                      signal12 := "BK12"."X14-2.ANODE NG P&P DOWN",
                      signal13 := "BK12"."X15-2.SPARE",
                      signal14 := "BK12"."X16-2.ANODE NG P&P ELECTRODE DETECT SENSOR",
                      signal15 := "BK12"."X17-2.SPARE",
                      interfaceSignals := #statInterfaceSignalsHmi[15].valueSymbolLeft,
                      ENO => #_w1);
   IF #_w1 THEN
       #instSignals15Right(interfaceSignals := #statInterfaceSignalsHmi[15].valueSymbolRight);   // "LAF_InterfaceSignalsBool"
   END_IF;
END_REGION

REGION Network 21: Interface Signals 05 -Example: Model Flex-Pro-Line - IN/OUT- / Interface Signals 16
   // Aufruf des Schnittstellen Signal Bausteins Ba-Bereich 4 / Call the interface signals bool blocks of opmode 4
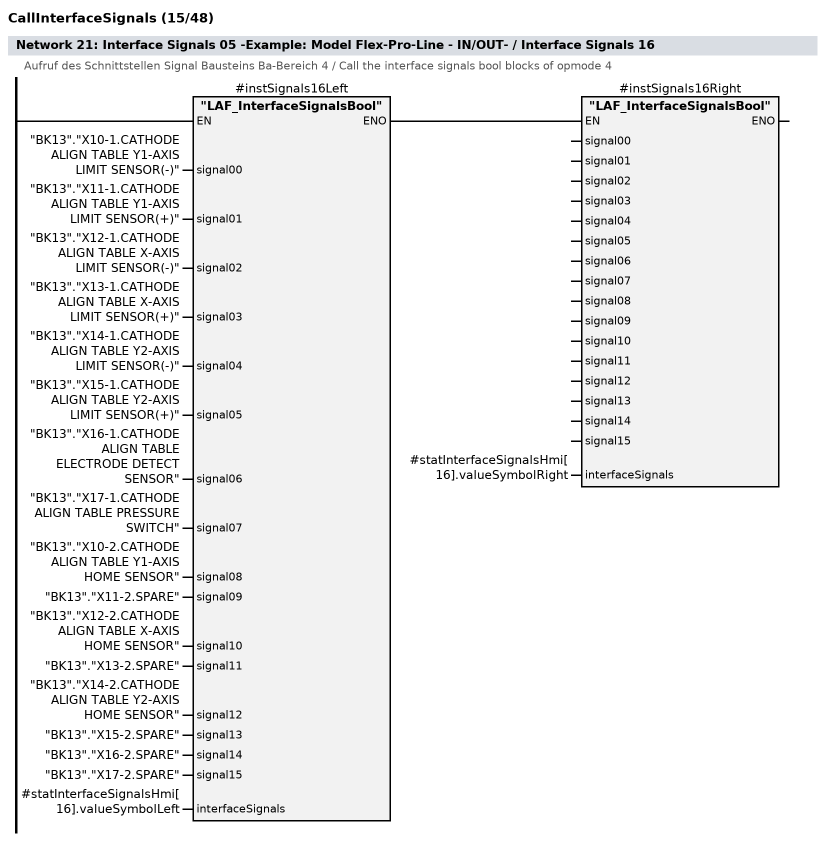
   RUNG wire#powerrail
      #instSignals16Left(signal00 := "BK13"."X10-1.CATHODE ALIGN TABLE Y1-AXIS LIMIT SENSOR(-)", signal01 := "BK13"."X11-1.CATHODE ALIGN TABLE Y1-AXIS LIMIT SENSOR(+)", signal02 := "BK13"."X12-1.CATHODE ALIGN TABLE X-AXIS LIMIT SENSOR(-)", signal03 := "BK13"."X13-1.CATHODE ALIGN TABLE X-AXIS LIMIT SENSOR(+)", signal04 := "BK13"."X14-1.CATHODE ALIGN TABLE Y2-AXIS LIMIT SENSOR(-)", signal05 := "BK13"."X15-1.CATHODE ALIGN TABLE Y2-AXIS LIMIT SENSOR(+)", signal06 := "BK13"."X16-1.CATHODE ALIGN TABLE ELECTRODE DETECT SENSOR", signal07 := "BK13"."X17-1.CATHODE ALIGN TABLE PRESSURE SWITCH", signal08 := "BK13"."X10-2.CATHODE ALIGN TABLE Y1-AXIS HOME SENSOR", signal09 := "BK13"."X11-2.SPARE", signal10 := "BK13"."X12-2.CATHODE ALIGN TABLE X-AXIS HOME SENSOR", signal11 := "BK13"."X13-2.SPARE", signal12 := "BK13"."X14-2.CATHODE ALIGN TABLE Y2-AXIS HOME SENSOR", signal13 := "BK13"."X15-2.SPARE", signal14 := "BK13"."X16-2.SPARE", signal15 := "BK13"."X17-2.SPARE", interfaceSignals := #statInterfaceSignalsHmi[16].valueSymbolLeft)
      #instSignals16Right(signal00 :=, signal01 :=, signal02 :=, signal03 :=, signal04 :=, signal05 :=, signal06 :=, signal07 :=, signal08 :=, signal09 :=, signal10 :=, signal11 :=, signal12 :=, signal13 :=, signal14 :=, signal15 :=, interfaceSignals := #statInterfaceSignalsHmi[16].valueSymbolRight)
   END_RUNG
   // the same network as SCL:
   #instSignals16Left(signal00 := "BK13"."X10-1.CATHODE ALIGN TABLE Y1-AXIS LIMIT SENSOR(-)",   // "LAF_InterfaceSignalsBool"
                      signal01 := "BK13"."X11-1.CATHODE ALIGN TABLE Y1-AXIS LIMIT SENSOR(+)",
                      signal02 := "BK13"."X12-1.CATHODE ALIGN TABLE X-AXIS LIMIT SENSOR(-)",
                      signal03 := "BK13"."X13-1.CATHODE ALIGN TABLE X-AXIS LIMIT SENSOR(+)",
                      signal04 := "BK13"."X14-1.CATHODE ALIGN TABLE Y2-AXIS LIMIT SENSOR(-)",
                      signal05 := "BK13"."X15-1.CATHODE ALIGN TABLE Y2-AXIS LIMIT SENSOR(+)",
                      signal06 := "BK13"."X16-1.CATHODE ALIGN TABLE ELECTRODE DETECT SENSOR",
                      signal07 := "BK13"."X17-1.CATHODE ALIGN TABLE PRESSURE SWITCH",
                      signal08 := "BK13"."X10-2.CATHODE ALIGN TABLE Y1-AXIS HOME SENSOR",
                      signal09 := "BK13"."X11-2.SPARE",
                      signal10 := "BK13"."X12-2.CATHODE ALIGN TABLE X-AXIS HOME SENSOR",
                      signal11 := "BK13"."X13-2.SPARE",
                      signal12 := "BK13"."X14-2.CATHODE ALIGN TABLE Y2-AXIS HOME SENSOR",
                      signal13 := "BK13"."X15-2.SPARE",
                      signal14 := "BK13"."X16-2.SPARE",
                      signal15 := "BK13"."X17-2.SPARE",
                      interfaceSignals := #statInterfaceSignalsHmi[16].valueSymbolLeft,
                      ENO => #_w1);
   IF #_w1 THEN
       #instSignals16Right(interfaceSignals := #statInterfaceSignalsHmi[16].valueSymbolRight);   // "LAF_InterfaceSignalsBool"
   END_IF;
END_REGION

REGION Network 22: Interface Signals 05 -Example: Model Flex-Pro-Line - IN/OUT- / Interface Signals 17
   // Aufruf des Schnittstellen Signal Bausteins Ba-Bereich 4 / Call the interface signals bool blocks of opmode 4
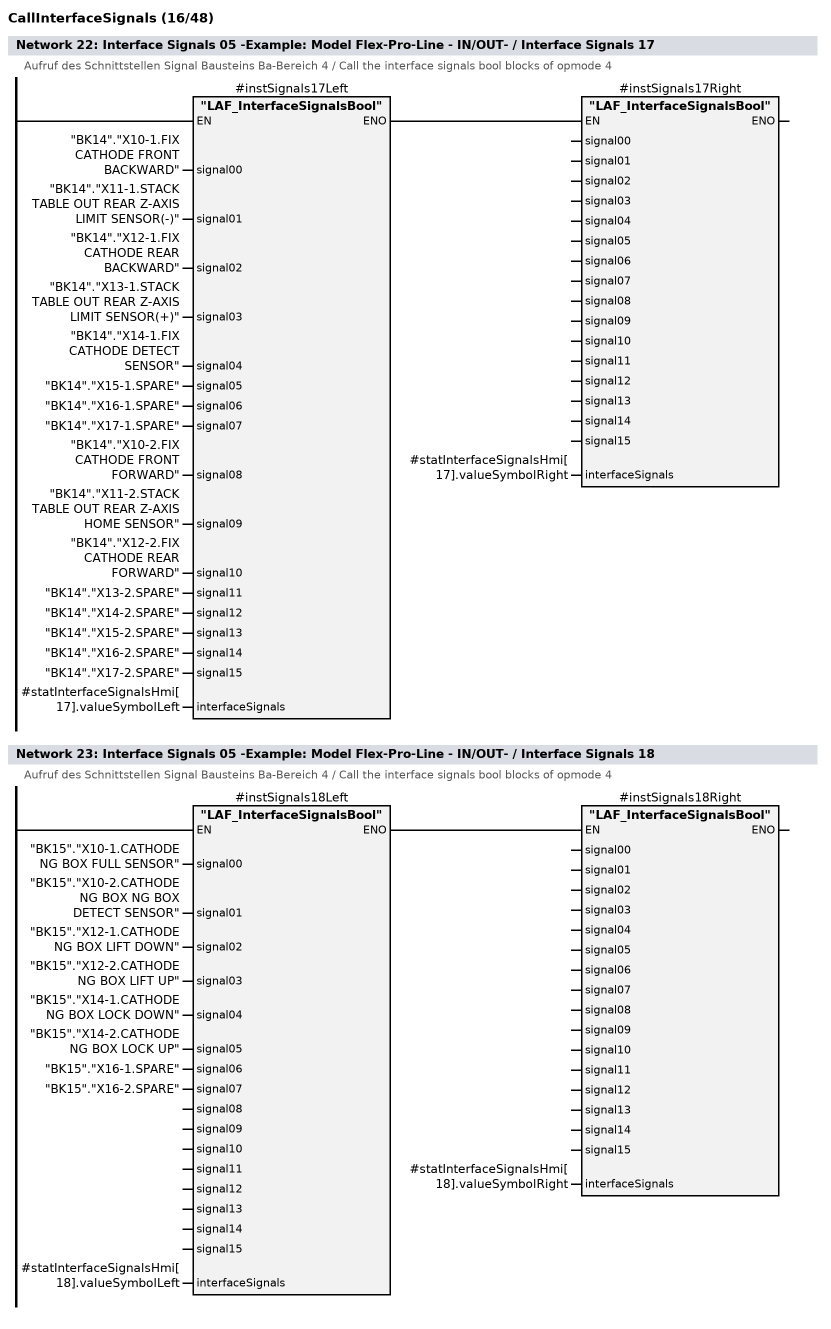
   RUNG wire#powerrail
      #instSignals17Left(signal00 := "BK14"."X10-1.FIX CATHODE FRONT BACKWARD", signal01 := "BK14"."X11-1.STACK TABLE OUT REAR Z-AXIS LIMIT SENSOR(-)", signal02 := "BK14"."X12-1.FIX CATHODE REAR BACKWARD", signal03 := "BK14"."X13-1.STACK TABLE OUT REAR Z-AXIS LIMIT SENSOR(+)", signal04 := "BK14"."X14-1.FIX CATHODE DETECT SENSOR", signal05 := "BK14"."X15-1.SPARE", signal06 := "BK14"."X16-1.SPARE", signal07 := "BK14"."X17-1.SPARE", signal08 := "BK14"."X10-2.FIX CATHODE FRONT FORWARD", signal09 := "BK14"."X11-2.STACK TABLE OUT REAR Z-AXIS HOME SENSOR", signal10 := "BK14"."X12-2.FIX CATHODE REAR FORWARD", signal11 := "BK14"."X13-2.SPARE", signal12 := "BK14"."X14-2.SPARE", signal13 := "BK14"."X15-2.SPARE", signal14 := "BK14"."X16-2.SPARE", signal15 := "BK14"."X17-2.SPARE", interfaceSignals := #statInterfaceSignalsHmi[17].valueSymbolLeft)
      #instSignals17Right(signal00 :=, signal01 :=, signal02 :=, signal03 :=, signal04 :=, signal05 :=, signal06 :=, signal07 :=, signal08 :=, signal09 :=, signal10 :=, signal11 :=, signal12 :=, signal13 :=, signal14 :=, signal15 :=, interfaceSignals := #statInterfaceSignalsHmi[17].valueSymbolRight)
   END_RUNG
   // the same network as SCL:
   #instSignals17Left(signal00 := "BK14"."X10-1.FIX CATHODE FRONT BACKWARD",   // "LAF_InterfaceSignalsBool"
                      signal01 := "BK14"."X11-1.STACK TABLE OUT REAR Z-AXIS LIMIT SENSOR(-)",
                      signal02 := "BK14"."X12-1.FIX CATHODE REAR BACKWARD",
                      signal03 := "BK14"."X13-1.STACK TABLE OUT REAR Z-AXIS LIMIT SENSOR(+)",
                      signal04 := "BK14"."X14-1.FIX CATHODE DETECT SENSOR",
                      signal05 := "BK14"."X15-1.SPARE",
                      signal06 := "BK14"."X16-1.SPARE",
                      signal07 := "BK14"."X17-1.SPARE",
                      signal08 := "BK14"."X10-2.FIX CATHODE FRONT FORWARD",
                      signal09 := "BK14"."X11-2.STACK TABLE OUT REAR Z-AXIS HOME SENSOR",
                      signal10 := "BK14"."X12-2.FIX CATHODE REAR FORWARD",
                      signal11 := "BK14"."X13-2.SPARE",
                      signal12 := "BK14"."X14-2.SPARE",
                      signal13 := "BK14"."X15-2.SPARE",
                      signal14 := "BK14"."X16-2.SPARE",
                      signal15 := "BK14"."X17-2.SPARE",
                      interfaceSignals := #statInterfaceSignalsHmi[17].valueSymbolLeft,
                      ENO => #_w1);
   IF #_w1 THEN
       #instSignals17Right(interfaceSignals := #statInterfaceSignalsHmi[17].valueSymbolRight);   // "LAF_InterfaceSignalsBool"
   END_IF;
END_REGION

REGION Network 23: Interface Signals 05 -Example: Model Flex-Pro-Line - IN/OUT- / Interface Signals 18
   // Aufruf des Schnittstellen Signal Bausteins Ba-Bereich 4 / Call the interface signals bool blocks of opmode 4
   RUNG wire#powerrail
      #instSignals18Left(signal00 := "BK15"."X10-1.CATHODE NG BOX FULL SENSOR", signal01 := "BK15"."X10-2.CATHODE NG BOX NG BOX DETECT SENSOR", signal02 := "BK15"."X12-1.CATHODE NG BOX LIFT DOWN", signal03 := "BK15"."X12-2.CATHODE NG BOX LIFT UP", signal04 := "BK15"."X14-1.CATHODE NG BOX LOCK DOWN", signal05 := "BK15"."X14-2.CATHODE NG BOX LOCK UP", signal06 := "BK15"."X16-1.SPARE", signal07 := "BK15"."X16-2.SPARE", signal08 :=, signal09 :=, signal10 :=, signal11 :=, signal12 :=, signal13 :=, signal14 :=, signal15 :=, interfaceSignals := #statInterfaceSignalsHmi[18].valueSymbolLeft)
      #instSignals18Right(signal00 :=, signal01 :=, signal02 :=, signal03 :=, signal04 :=, signal05 :=, signal06 :=, signal07 :=, signal08 :=, signal09 :=, signal10 :=, signal11 :=, signal12 :=, signal13 :=, signal14 :=, signal15 :=, interfaceSignals := #statInterfaceSignalsHmi[18].valueSymbolRight)
   END_RUNG
   // the same network as SCL:
   #instSignals18Left(signal00 := "BK15"."X10-1.CATHODE NG BOX FULL SENSOR",   // "LAF_InterfaceSignalsBool"
                      signal01 := "BK15"."X10-2.CATHODE NG BOX NG BOX DETECT SENSOR",
                      signal02 := "BK15"."X12-1.CATHODE NG BOX LIFT DOWN",
                      signal03 := "BK15"."X12-2.CATHODE NG BOX LIFT UP",
                      signal04 := "BK15"."X14-1.CATHODE NG BOX LOCK DOWN",
                      signal05 := "BK15"."X14-2.CATHODE NG BOX LOCK UP",
                      signal06 := "BK15"."X16-1.SPARE",
                      signal07 := "BK15"."X16-2.SPARE",
                      interfaceSignals := #statInterfaceSignalsHmi[18].valueSymbolLeft,
                      ENO => #_w1);
   IF #_w1 THEN
       #instSignals18Right(interfaceSignals := #statInterfaceSignalsHmi[18].valueSymbolRight);   // "LAF_InterfaceSignalsBool"
   END_IF;
END_REGION

REGION Network 24: Interface Signals 05 -Example: Model Flex-Pro-Line - IN/OUT- / Interface Signals 19
   // Aufruf des Schnittstellen Signal Bausteins Ba-Bereich 4 / Call the interface signals bool blocks of opmode 4
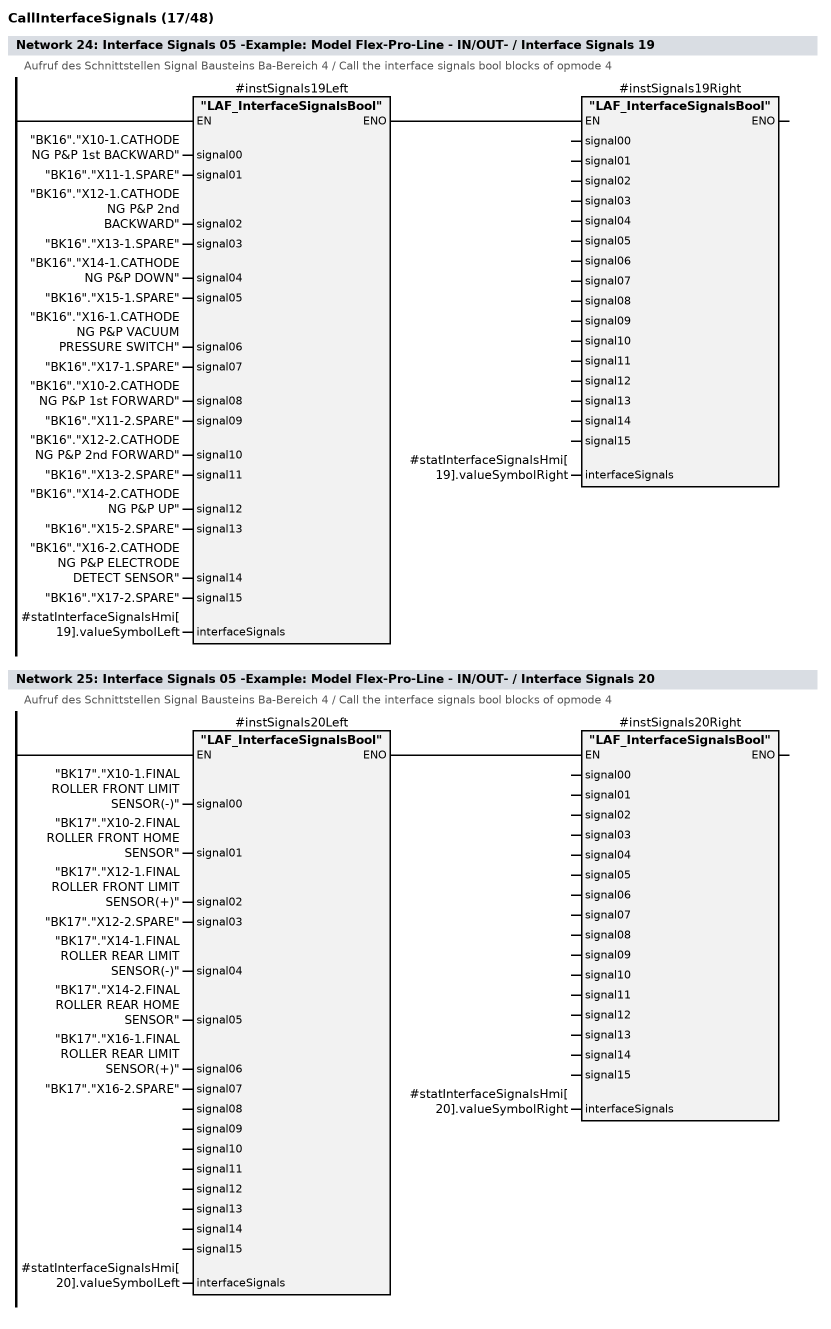
   RUNG wire#powerrail
      #instSignals19Left(signal00 := "BK16"."X10-1.CATHODE NG P&P 1st BACKWARD", signal01 := "BK16"."X11-1.SPARE", signal02 := "BK16"."X12-1.CATHODE NG P&P 2nd BACKWARD", signal03 := "BK16"."X13-1.SPARE", signal04 := "BK16"."X14-1.CATHODE NG P&P DOWN", signal05 := "BK16"."X15-1.SPARE", signal06 := "BK16"."X16-1.CATHODE NG P&P VACUUM PRESSURE SWITCH", signal07 := "BK16"."X17-1.SPARE", signal08 := "BK16"."X10-2.CATHODE NG P&P 1st FORWARD", signal09 := "BK16"."X11-2.SPARE", signal10 := "BK16"."X12-2.CATHODE NG P&P 2nd FORWARD", signal11 := "BK16"."X13-2.SPARE", signal12 := "BK16"."X14-2.CATHODE NG P&P UP", signal13 := "BK16"."X15-2.SPARE", signal14 := "BK16"."X16-2.CATHODE NG P&P ELECTRODE DETECT SENSOR", signal15 := "BK16"."X17-2.SPARE", interfaceSignals := #statInterfaceSignalsHmi[19].valueSymbolLeft)
      #instSignals19Right(signal00 :=, signal01 :=, signal02 :=, signal03 :=, signal04 :=, signal05 :=, signal06 :=, signal07 :=, signal08 :=, signal09 :=, signal10 :=, signal11 :=, signal12 :=, signal13 :=, signal14 :=, signal15 :=, interfaceSignals := #statInterfaceSignalsHmi[19].valueSymbolRight)
   END_RUNG
   // the same network as SCL:
   #instSignals19Left(signal00 := "BK16"."X10-1.CATHODE NG P&P 1st BACKWARD",   // "LAF_InterfaceSignalsBool"
                      signal01 := "BK16"."X11-1.SPARE",
                      signal02 := "BK16"."X12-1.CATHODE NG P&P 2nd BACKWARD",
                      signal03 := "BK16"."X13-1.SPARE",
                      signal04 := "BK16"."X14-1.CATHODE NG P&P DOWN",
                      signal05 := "BK16"."X15-1.SPARE",
                      signal06 := "BK16"."X16-1.CATHODE NG P&P VACUUM PRESSURE SWITCH",
                      signal07 := "BK16"."X17-1.SPARE",
                      signal08 := "BK16"."X10-2.CATHODE NG P&P 1st FORWARD",
                      signal09 := "BK16"."X11-2.SPARE",
                      signal10 := "BK16"."X12-2.CATHODE NG P&P 2nd FORWARD",
                      signal11 := "BK16"."X13-2.SPARE",
                      signal12 := "BK16"."X14-2.CATHODE NG P&P UP",
                      signal13 := "BK16"."X15-2.SPARE",
                      signal14 := "BK16"."X16-2.CATHODE NG P&P ELECTRODE DETECT SENSOR",
                      signal15 := "BK16"."X17-2.SPARE",
                      interfaceSignals := #statInterfaceSignalsHmi[19].valueSymbolLeft,
                      ENO => #_w1);
   IF #_w1 THEN
       #instSignals19Right(interfaceSignals := #statInterfaceSignalsHmi[19].valueSymbolRight);   // "LAF_InterfaceSignalsBool"
   END_IF;
END_REGION

REGION Network 25: Interface Signals 05 -Example: Model Flex-Pro-Line - IN/OUT- / Interface Signals 20
   // Aufruf des Schnittstellen Signal Bausteins Ba-Bereich 4 / Call the interface signals bool blocks of opmode 4
   RUNG wire#powerrail
      #instSignals20Left(signal00 := "BK17"."X10-1.FINAL ROLLER FRONT LIMIT SENSOR(-)", signal01 := "BK17"."X10-2.FINAL ROLLER FRONT HOME SENSOR", signal02 := "BK17"."X12-1.FINAL ROLLER FRONT LIMIT SENSOR(+)", signal03 := "BK17"."X12-2.SPARE", signal04 := "BK17"."X14-1.FINAL ROLLER REAR LIMIT SENSOR(-)", signal05 := "BK17"."X14-2.FINAL ROLLER REAR HOME SENSOR", signal06 := "BK17"."X16-1.FINAL ROLLER REAR LIMIT SENSOR(+)", signal07 := "BK17"."X16-2.SPARE", signal08 :=, signal09 :=, signal10 :=, signal11 :=, signal12 :=, signal13 :=, signal14 :=, signal15 :=, interfaceSignals := #statInterfaceSignalsHmi[20].valueSymbolLeft)
      #instSignals20Right(signal00 :=, signal01 :=, signal02 :=, signal03 :=, signal04 :=, signal05 :=, signal06 :=, signal07 :=, signal08 :=, signal09 :=, signal10 :=, signal11 :=, signal12 :=, signal13 :=, signal14 :=, signal15 :=, interfaceSignals := #statInterfaceSignalsHmi[20].valueSymbolRight)
   END_RUNG
   // the same network as SCL:
   #instSignals20Left(signal00 := "BK17"."X10-1.FINAL ROLLER FRONT LIMIT SENSOR(-)",   // "LAF_InterfaceSignalsBool"
                      signal01 := "BK17"."X10-2.FINAL ROLLER FRONT HOME SENSOR",
                      signal02 := "BK17"."X12-1.FINAL ROLLER FRONT LIMIT SENSOR(+)",
                      signal03 := "BK17"."X12-2.SPARE",
                      signal04 := "BK17"."X14-1.FINAL ROLLER REAR LIMIT SENSOR(-)",
                      signal05 := "BK17"."X14-2.FINAL ROLLER REAR HOME SENSOR",
                      signal06 := "BK17"."X16-1.FINAL ROLLER REAR LIMIT SENSOR(+)",
                      signal07 := "BK17"."X16-2.SPARE",
                      interfaceSignals := #statInterfaceSignalsHmi[20].valueSymbolLeft,
                      ENO => #_w1);
   IF #_w1 THEN
       #instSignals20Right(interfaceSignals := #statInterfaceSignalsHmi[20].valueSymbolRight);   // "LAF_InterfaceSignalsBool"
   END_IF;
END_REGION

REGION Network 26: Interface Signals 05 -Example: Model Flex-Pro-Line - IN/OUT- / Interface Signals 21
   // Aufruf des Schnittstellen Signal Bausteins Ba-Bereich 4 / Call the interface signals bool blocks of opmode 4
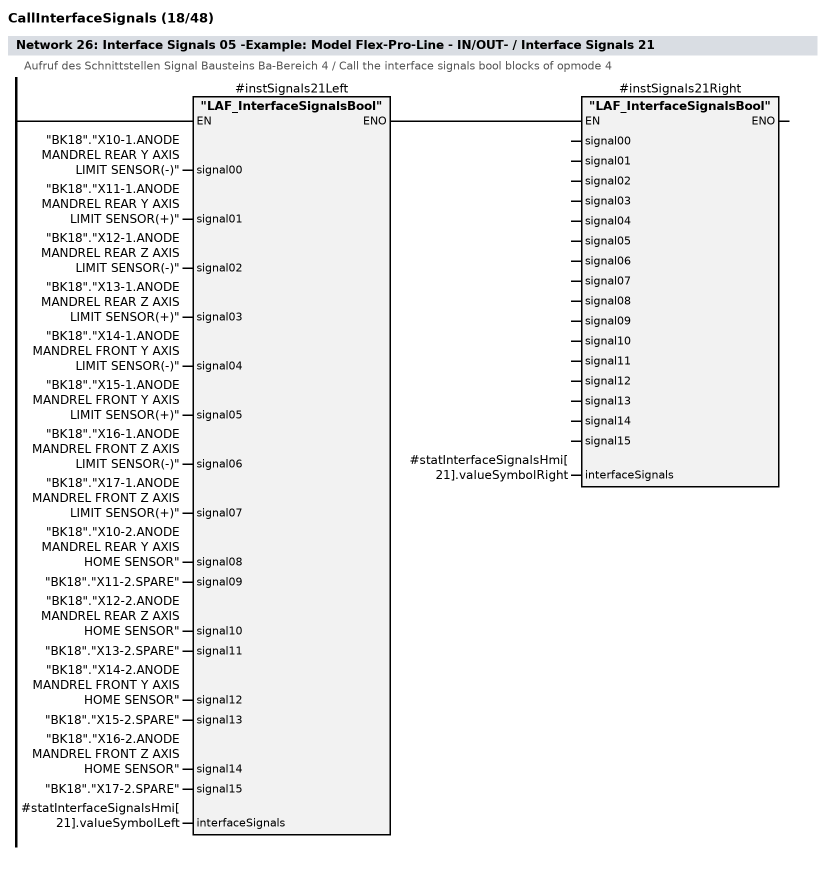
   RUNG wire#powerrail
      #instSignals21Left(signal00 := "BK18"."X10-1.ANODE MANDREL REAR Y AXIS LIMIT SENSOR(-)", signal01 := "BK18"."X11-1.ANODE MANDREL REAR Y AXIS LIMIT SENSOR(+)", signal02 := "BK18"."X12-1.ANODE MANDREL REAR Z AXIS LIMIT SENSOR(-)", signal03 := "BK18"."X13-1.ANODE MANDREL REAR Z AXIS LIMIT SENSOR(+)", signal04 := "BK18"."X14-1.ANODE MANDREL FRONT Y AXIS LIMIT SENSOR(-)", signal05 := "BK18"."X15-1.ANODE MANDREL FRONT Y AXIS LIMIT SENSOR(+)", signal06 := "BK18"."X16-1.ANODE MANDREL FRONT Z AXIS LIMIT SENSOR(-)", signal07 := "BK18"."X17-1.ANODE MANDREL FRONT Z AXIS LIMIT SENSOR(+)", signal08 := "BK18"."X10-2.ANODE MANDREL REAR Y AXIS HOME SENSOR", signal09 := "BK18"."X11-2.SPARE", signal10 := "BK18"."X12-2.ANODE MANDREL REAR Z AXIS HOME SENSOR", signal11 := "BK18"."X13-2.SPARE", signal12 := "BK18"."X14-2.ANODE MANDREL FRONT Y AXIS HOME SENSOR", signal13 := "BK18"."X15-2.SPARE", signal14 := "BK18"."X16-2.ANODE MANDREL FRONT Z AXIS HOME SENSOR", signal15 := "BK18"."X17-2.SPARE", interfaceSignals := #statInterfaceSignalsHmi[21].valueSymbolLeft)
      #instSignals21Right(signal00 :=, signal01 :=, signal02 :=, signal03 :=, signal04 :=, signal05 :=, signal06 :=, signal07 :=, signal08 :=, signal09 :=, signal10 :=, signal11 :=, signal12 :=, signal13 :=, signal14 :=, signal15 :=, interfaceSignals := #statInterfaceSignalsHmi[21].valueSymbolRight)
   END_RUNG
   // the same network as SCL:
   #instSignals21Left(signal00 := "BK18"."X10-1.ANODE MANDREL REAR Y AXIS LIMIT SENSOR(-)",   // "LAF_InterfaceSignalsBool"
                      signal01 := "BK18"."X11-1.ANODE MANDREL REAR Y AXIS LIMIT SENSOR(+)",
                      signal02 := "BK18"."X12-1.ANODE MANDREL REAR Z AXIS LIMIT SENSOR(-)",
                      signal03 := "BK18"."X13-1.ANODE MANDREL REAR Z AXIS LIMIT SENSOR(+)",
                      signal04 := "BK18"."X14-1.ANODE MANDREL FRONT Y AXIS LIMIT SENSOR(-)",
                      signal05 := "BK18"."X15-1.ANODE MANDREL FRONT Y AXIS LIMIT SENSOR(+)",
                      signal06 := "BK18"."X16-1.ANODE MANDREL FRONT Z AXIS LIMIT SENSOR(-)",
                      signal07 := "BK18"."X17-1.ANODE MANDREL FRONT Z AXIS LIMIT SENSOR(+)",
                      signal08 := "BK18"."X10-2.ANODE MANDREL REAR Y AXIS HOME SENSOR",
                      signal09 := "BK18"."X11-2.SPARE",
                      signal10 := "BK18"."X12-2.ANODE MANDREL REAR Z AXIS HOME SENSOR",
                      signal11 := "BK18"."X13-2.SPARE",
                      signal12 := "BK18"."X14-2.ANODE MANDREL FRONT Y AXIS HOME SENSOR",
                      signal13 := "BK18"."X15-2.SPARE",
                      signal14 := "BK18"."X16-2.ANODE MANDREL FRONT Z AXIS HOME SENSOR",
                      signal15 := "BK18"."X17-2.SPARE",
                      interfaceSignals := #statInterfaceSignalsHmi[21].valueSymbolLeft,
                      ENO => #_w1);
   IF #_w1 THEN
       #instSignals21Right(interfaceSignals := #statInterfaceSignalsHmi[21].valueSymbolRight);   // "LAF_InterfaceSignalsBool"
   END_IF;
END_REGION

REGION Network 27: Interface Signals 05 -Example: Model Flex-Pro-Line - IN/OUT- / Interface Signals 22
   // Aufruf des Schnittstellen Signal Bausteins Ba-Bereich 4 / Call the interface signals bool blocks of opmode 4
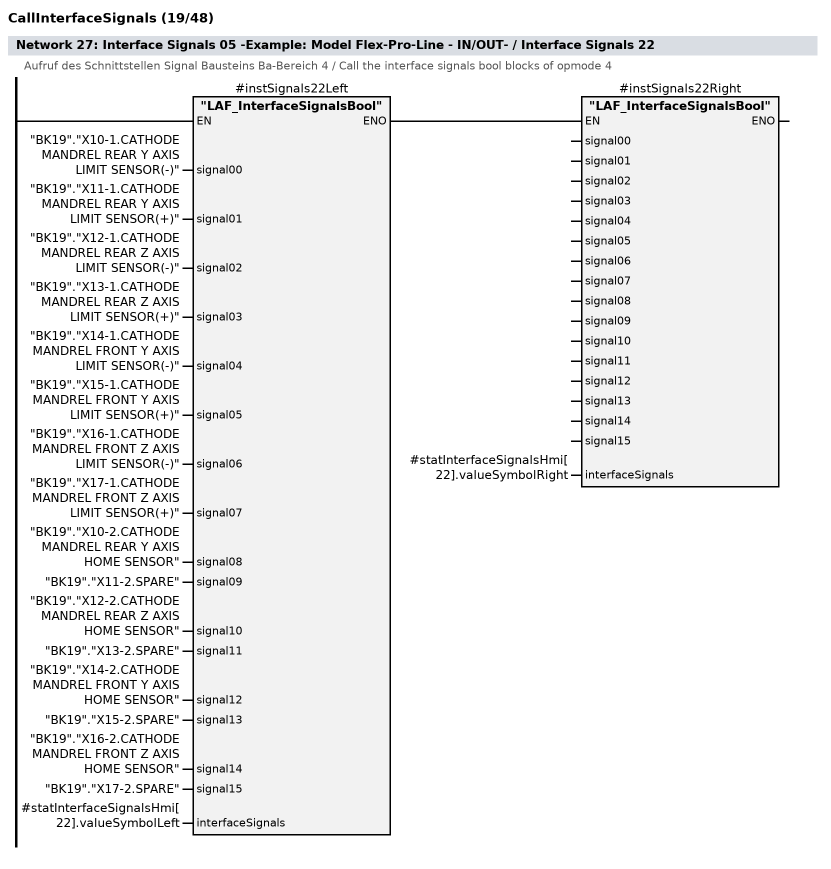
   RUNG wire#powerrail
      #instSignals22Left(signal00 := "BK19"."X10-1.CATHODE MANDREL REAR Y AXIS LIMIT SENSOR(-)", signal01 := "BK19"."X11-1.CATHODE MANDREL REAR Y AXIS LIMIT SENSOR(+)", signal02 := "BK19"."X12-1.CATHODE MANDREL REAR Z AXIS LIMIT SENSOR(-)", signal03 := "BK19"."X13-1.CATHODE MANDREL REAR Z AXIS LIMIT SENSOR(+)", signal04 := "BK19"."X14-1.CATHODE MANDREL FRONT Y AXIS LIMIT SENSOR(-)", signal05 := "BK19"."X15-1.CATHODE MANDREL FRONT Y AXIS LIMIT SENSOR(+)", signal06 := "BK19"."X16-1.CATHODE MANDREL FRONT Z AXIS LIMIT SENSOR(-)", signal07 := "BK19"."X17-1.CATHODE MANDREL FRONT Z AXIS LIMIT SENSOR(+)", signal08 := "BK19"."X10-2.CATHODE MANDREL REAR Y AXIS HOME SENSOR", signal09 := "BK19"."X11-2.SPARE", signal10 := "BK19"."X12-2.CATHODE MANDREL REAR Z AXIS HOME SENSOR", signal11 := "BK19"."X13-2.SPARE", signal12 := "BK19"."X14-2.CATHODE MANDREL FRONT Y AXIS HOME SENSOR", signal13 := "BK19"."X15-2.SPARE", signal14 := "BK19"."X16-2.CATHODE MANDREL FRONT Z AXIS HOME SENSOR", signal15 := "BK19"."X17-2.SPARE", interfaceSignals := #statInterfaceSignalsHmi[22].valueSymbolLeft)
      #instSignals22Right(signal00 :=, signal01 :=, signal02 :=, signal03 :=, signal04 :=, signal05 :=, signal06 :=, signal07 :=, signal08 :=, signal09 :=, signal10 :=, signal11 :=, signal12 :=, signal13 :=, signal14 :=, signal15 :=, interfaceSignals := #statInterfaceSignalsHmi[22].valueSymbolRight)
   END_RUNG
   // the same network as SCL:
   #instSignals22Left(signal00 := "BK19"."X10-1.CATHODE MANDREL REAR Y AXIS LIMIT SENSOR(-)",   // "LAF_InterfaceSignalsBool"
                      signal01 := "BK19"."X11-1.CATHODE MANDREL REAR Y AXIS LIMIT SENSOR(+)",
                      signal02 := "BK19"."X12-1.CATHODE MANDREL REAR Z AXIS LIMIT SENSOR(-)",
                      signal03 := "BK19"."X13-1.CATHODE MANDREL REAR Z AXIS LIMIT SENSOR(+)",
                      signal04 := "BK19"."X14-1.CATHODE MANDREL FRONT Y AXIS LIMIT SENSOR(-)",
                      signal05 := "BK19"."X15-1.CATHODE MANDREL FRONT Y AXIS LIMIT SENSOR(+)",
                      signal06 := "BK19"."X16-1.CATHODE MANDREL FRONT Z AXIS LIMIT SENSOR(-)",
                      signal07 := "BK19"."X17-1.CATHODE MANDREL FRONT Z AXIS LIMIT SENSOR(+)",
                      signal08 := "BK19"."X10-2.CATHODE MANDREL REAR Y AXIS HOME SENSOR",
                      signal09 := "BK19"."X11-2.SPARE",
                      signal10 := "BK19"."X12-2.CATHODE MANDREL REAR Z AXIS HOME SENSOR",
                      signal11 := "BK19"."X13-2.SPARE",
                      signal12 := "BK19"."X14-2.CATHODE MANDREL FRONT Y AXIS HOME SENSOR",
                      signal13 := "BK19"."X15-2.SPARE",
                      signal14 := "BK19"."X16-2.CATHODE MANDREL FRONT Z AXIS HOME SENSOR",
                      signal15 := "BK19"."X17-2.SPARE",
                      interfaceSignals := #statInterfaceSignalsHmi[22].valueSymbolLeft,
                      ENO => #_w1);
   IF #_w1 THEN
       #instSignals22Right(interfaceSignals := #statInterfaceSignalsHmi[22].valueSymbolRight);   // "LAF_InterfaceSignalsBool"
   END_IF;
END_REGION

REGION Network 28: Interface Signals 03 -Example: System flags & Clock flags- / Interface Signals23
   // Aufruf des Schnittstellen Signal Bausteins für die Systemvariablen / Call the interface signals bool blocks of system tags
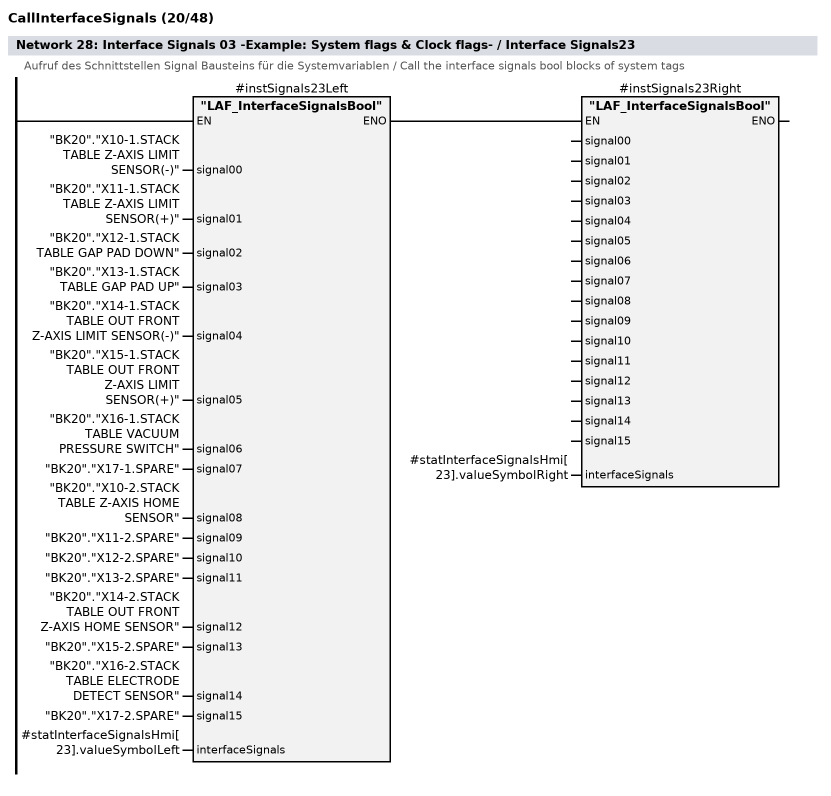
   RUNG wire#powerrail
      #instSignals23Left(signal00 := "BK20"."X10-1.STACK TABLE Z-AXIS LIMIT SENSOR(-)", signal01 := "BK20"."X11-1.STACK TABLE Z-AXIS LIMIT SENSOR(+)", signal02 := "BK20"."X12-1.STACK TABLE GAP PAD DOWN", signal03 := "BK20"."X13-1.STACK TABLE GAP PAD UP", signal04 := "BK20"."X14-1.STACK TABLE OUT FRONT Z-AXIS LIMIT SENSOR(-)", signal05 := "BK20"."X15-1.STACK TABLE OUT FRONT Z-AXIS LIMIT SENSOR(+)", signal06 := "BK20"."X16-1.STACK TABLE VACUUM PRESSURE SWITCH", signal07 := "BK20"."X17-1.SPARE", signal08 := "BK20"."X10-2.STACK TABLE Z-AXIS HOME SENSOR", signal09 := "BK20"."X11-2.SPARE", signal10 := "BK20"."X12-2.SPARE", signal11 := "BK20"."X13-2.SPARE", signal12 := "BK20"."X14-2.STACK TABLE OUT FRONT Z-AXIS HOME SENSOR", signal13 := "BK20"."X15-2.SPARE", signal14 := "BK20"."X16-2.STACK TABLE ELECTRODE DETECT SENSOR", signal15 := "BK20"."X17-2.SPARE", interfaceSignals := #statInterfaceSignalsHmi[23].valueSymbolLeft)
      #instSignals23Right(signal00 :=, signal01 :=, signal02 :=, signal03 :=, signal04 :=, signal05 :=, signal06 :=, signal07 :=, signal08 :=, signal09 :=, signal10 :=, signal11 :=, signal12 :=, signal13 :=, signal14 :=, signal15 :=, interfaceSignals := #statInterfaceSignalsHmi[23].valueSymbolRight)
   END_RUNG
   // the same network as SCL:
   #instSignals23Left(signal00 := "BK20"."X10-1.STACK TABLE Z-AXIS LIMIT SENSOR(-)",   // "LAF_InterfaceSignalsBool"
                      signal01 := "BK20"."X11-1.STACK TABLE Z-AXIS LIMIT SENSOR(+)",
                      signal02 := "BK20"."X12-1.STACK TABLE GAP PAD DOWN",
                      signal03 := "BK20"."X13-1.STACK TABLE GAP PAD UP",
                      signal04 := "BK20"."X14-1.STACK TABLE OUT FRONT Z-AXIS LIMIT SENSOR(-)",
                      signal05 := "BK20"."X15-1.STACK TABLE OUT FRONT Z-AXIS LIMIT SENSOR(+)",
                      signal06 := "BK20"."X16-1.STACK TABLE VACUUM PRESSURE SWITCH",
                      signal07 := "BK20"."X17-1.SPARE",
                      signal08 := "BK20"."X10-2.STACK TABLE Z-AXIS HOME SENSOR",
                      signal09 := "BK20"."X11-2.SPARE",
                      signal10 := "BK20"."X12-2.SPARE",
                      signal11 := "BK20"."X13-2.SPARE",
                      signal12 := "BK20"."X14-2.STACK TABLE OUT FRONT Z-AXIS HOME SENSOR",
                      signal13 := "BK20"."X15-2.SPARE",
                      signal14 := "BK20"."X16-2.STACK TABLE ELECTRODE DETECT SENSOR",
                      signal15 := "BK20"."X17-2.SPARE",
                      interfaceSignals := #statInterfaceSignalsHmi[23].valueSymbolLeft,
                      ENO => #_w1);
   IF #_w1 THEN
       #instSignals23Right(interfaceSignals := #statInterfaceSignalsHmi[23].valueSymbolRight);   // "LAF_InterfaceSignalsBool"
   END_IF;
END_REGION

REGION Network 29: Interface Signals 04 -Example: Model Flex-Pro-Line - IN/OUT- / Interface Signals 24
   // Aufruf des Schnittstellen Signal Bausteins Ba-Bereich 4 / Call the interface signals bool blocks of opmode 4
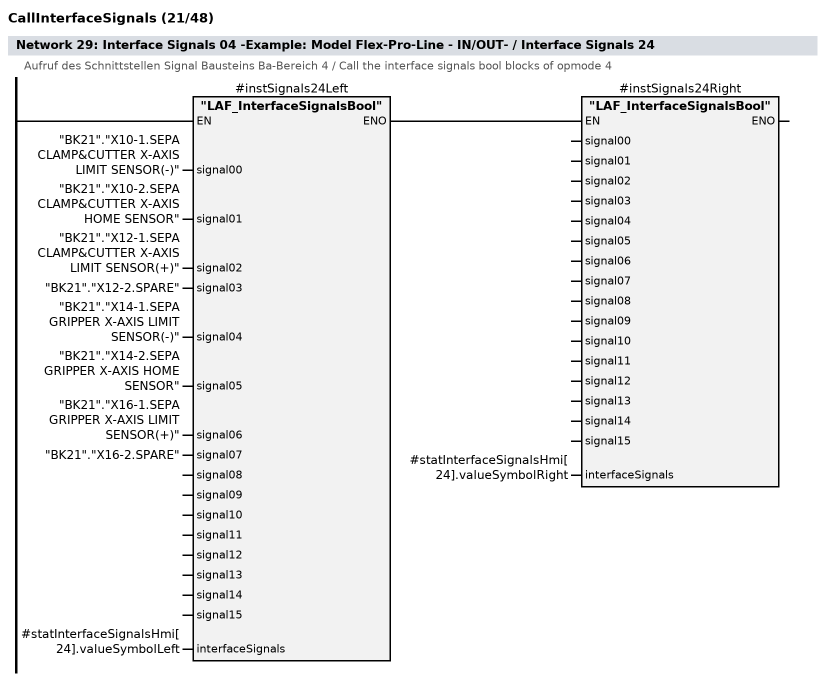
   RUNG wire#powerrail
      #instSignals24Left(signal00 := "BK21"."X10-1.SEPA CLAMP&CUTTER X-AXIS LIMIT SENSOR(-)", signal01 := "BK21"."X10-2.SEPA CLAMP&CUTTER X-AXIS HOME SENSOR", signal02 := "BK21"."X12-1.SEPA CLAMP&CUTTER X-AXIS LIMIT SENSOR(+)", signal03 := "BK21"."X12-2.SPARE", signal04 := "BK21"."X14-1.SEPA GRIPPER X-AXIS LIMIT SENSOR(-)", signal05 := "BK21"."X14-2.SEPA GRIPPER X-AXIS HOME SENSOR", signal06 := "BK21"."X16-1.SEPA GRIPPER X-AXIS LIMIT SENSOR(+)", signal07 := "BK21"."X16-2.SPARE", signal08 :=, signal09 :=, signal10 :=, signal11 :=, signal12 :=, signal13 :=, signal14 :=, signal15 :=, interfaceSignals := #statInterfaceSignalsHmi[24].valueSymbolLeft)
      #instSignals24Right(signal00 :=, signal01 :=, signal02 :=, signal03 :=, signal04 :=, signal05 :=, signal06 :=, signal07 :=, signal08 :=, signal09 :=, signal10 :=, signal11 :=, signal12 :=, signal13 :=, signal14 :=, signal15 :=, interfaceSignals := #statInterfaceSignalsHmi[24].valueSymbolRight)
   END_RUNG
   // the same network as SCL:
   #instSignals24Left(signal00 := "BK21"."X10-1.SEPA CLAMP&CUTTER X-AXIS LIMIT SENSOR(-)",   // "LAF_InterfaceSignalsBool"
                      signal01 := "BK21"."X10-2.SEPA CLAMP&CUTTER X-AXIS HOME SENSOR",
                      signal02 := "BK21"."X12-1.SEPA CLAMP&CUTTER X-AXIS LIMIT SENSOR(+)",
                      signal03 := "BK21"."X12-2.SPARE",
                      signal04 := "BK21"."X14-1.SEPA GRIPPER X-AXIS LIMIT SENSOR(-)",
                      signal05 := "BK21"."X14-2.SEPA GRIPPER X-AXIS HOME SENSOR",
                      signal06 := "BK21"."X16-1.SEPA GRIPPER X-AXIS LIMIT SENSOR(+)",
                      signal07 := "BK21"."X16-2.SPARE",
                      interfaceSignals := #statInterfaceSignalsHmi[24].valueSymbolLeft,
                      ENO => #_w1);
   IF #_w1 THEN
       #instSignals24Right(interfaceSignals := #statInterfaceSignalsHmi[24].valueSymbolRight);   // "LAF_InterfaceSignalsBool"
   END_IF;
END_REGION

REGION Network 30: Interface Signals 05 -Example: Model Flex-Pro-Line - IN/OUT- / Interface Signals 25
   // Aufruf des Schnittstellen Signal Bausteins Ba-Bereich 4 / Call the interface signals bool blocks of opmode 4
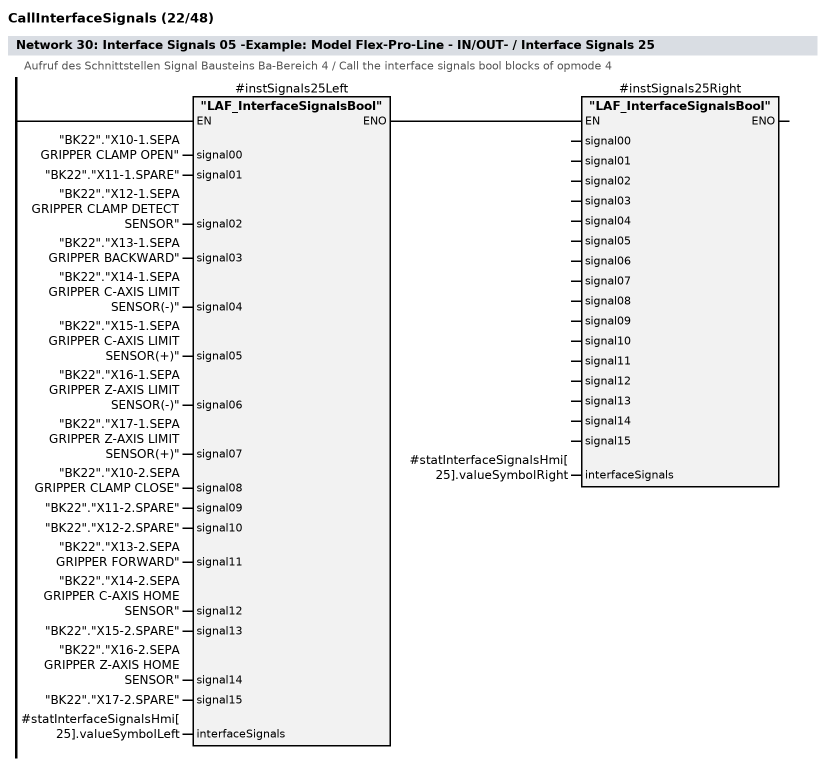
   RUNG wire#powerrail
      #instSignals25Left(signal00 := "BK22"."X10-1.SEPA GRIPPER CLAMP OPEN", signal01 := "BK22"."X11-1.SPARE", signal02 := "BK22"."X12-1.SEPA GRIPPER CLAMP DETECT SENSOR", signal03 := "BK22"."X13-1.SEPA GRIPPER BACKWARD", signal04 := "BK22"."X14-1.SEPA GRIPPER C-AXIS LIMIT SENSOR(-)", signal05 := "BK22"."X15-1.SEPA GRIPPER C-AXIS LIMIT SENSOR(+)", signal06 := "BK22"."X16-1.SEPA GRIPPER Z-AXIS LIMIT SENSOR(-)", signal07 := "BK22"."X17-1.SEPA GRIPPER Z-AXIS LIMIT SENSOR(+)", signal08 := "BK22"."X10-2.SEPA GRIPPER CLAMP CLOSE", signal09 := "BK22"."X11-2.SPARE", signal10 := "BK22"."X12-2.SPARE", signal11 := "BK22"."X13-2.SEPA GRIPPER FORWARD", signal12 := "BK22"."X14-2.SEPA GRIPPER C-AXIS HOME SENSOR", signal13 := "BK22"."X15-2.SPARE", signal14 := "BK22"."X16-2.SEPA GRIPPER Z-AXIS HOME SENSOR", signal15 := "BK22"."X17-2.SPARE", interfaceSignals := #statInterfaceSignalsHmi[25].valueSymbolLeft)
      #instSignals25Right(signal00 :=, signal01 :=, signal02 :=, signal03 :=, signal04 :=, signal05 :=, signal06 :=, signal07 :=, signal08 :=, signal09 :=, signal10 :=, signal11 :=, signal12 :=, signal13 :=, signal14 :=, signal15 :=, interfaceSignals := #statInterfaceSignalsHmi[25].valueSymbolRight)
   END_RUNG
   // the same network as SCL:
   #instSignals25Left(signal00 := "BK22"."X10-1.SEPA GRIPPER CLAMP OPEN",   // "LAF_InterfaceSignalsBool"
                      signal01 := "BK22"."X11-1.SPARE",
                      signal02 := "BK22"."X12-1.SEPA GRIPPER CLAMP DETECT SENSOR",
                      signal03 := "BK22"."X13-1.SEPA GRIPPER BACKWARD",
                      signal04 := "BK22"."X14-1.SEPA GRIPPER C-AXIS LIMIT SENSOR(-)",
                      signal05 := "BK22"."X15-1.SEPA GRIPPER C-AXIS LIMIT SENSOR(+)",
                      signal06 := "BK22"."X16-1.SEPA GRIPPER Z-AXIS LIMIT SENSOR(-)",
                      signal07 := "BK22"."X17-1.SEPA GRIPPER Z-AXIS LIMIT SENSOR(+)",
                      signal08 := "BK22"."X10-2.SEPA GRIPPER CLAMP CLOSE",
                      signal09 := "BK22"."X11-2.SPARE",
                      signal10 := "BK22"."X12-2.SPARE",
                      signal11 := "BK22"."X13-2.SEPA GRIPPER FORWARD",
                      signal12 := "BK22"."X14-2.SEPA GRIPPER C-AXIS HOME SENSOR",
                      signal13 := "BK22"."X15-2.SPARE",
                      signal14 := "BK22"."X16-2.SEPA GRIPPER Z-AXIS HOME SENSOR",
                      signal15 := "BK22"."X17-2.SPARE",
                      interfaceSignals := #statInterfaceSignalsHmi[25].valueSymbolLeft,
                      ENO => #_w1);
   IF #_w1 THEN
       #instSignals25Right(interfaceSignals := #statInterfaceSignalsHmi[25].valueSymbolRight);   // "LAF_InterfaceSignalsBool"
   END_IF;
END_REGION

REGION Network 31: Interface Signals 05 -Example: Model Flex-Pro-Line - IN/OUT- / Interface Signals 26
   // Aufruf des Schnittstellen Signal Bausteins Ba-Bereich 4 / Call the interface signals bool blocks of opmode 4
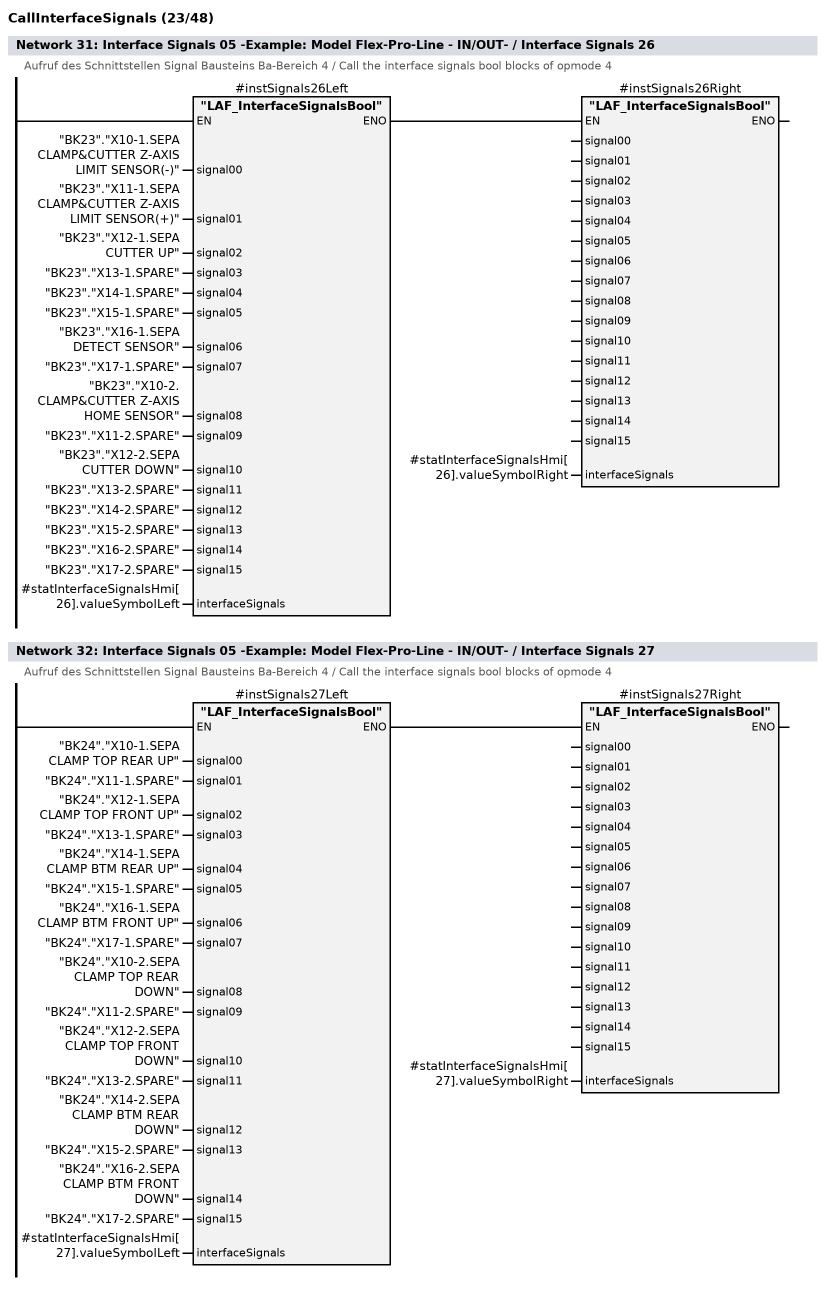
   RUNG wire#powerrail
      #instSignals26Left(signal00 := "BK23"."X10-1.SEPA CLAMP&CUTTER Z-AXIS LIMIT SENSOR(-)", signal01 := "BK23"."X11-1.SEPA CLAMP&CUTTER Z-AXIS LIMIT SENSOR(+)", signal02 := "BK23"."X12-1.SEPA CUTTER UP", signal03 := "BK23"."X13-1.SPARE", signal04 := "BK23"."X14-1.SPARE", signal05 := "BK23"."X15-1.SPARE", signal06 := "BK23"."X16-1.SEPA DETECT SENSOR", signal07 := "BK23"."X17-1.SPARE", signal08 := "BK23"."X10-2.CLAMP&CUTTER Z-AXIS HOME SENSOR", signal09 := "BK23"."X11-2.SPARE", signal10 := "BK23"."X12-2.SEPA CUTTER DOWN", signal11 := "BK23"."X13-2.SPARE", signal12 := "BK23"."X14-2.SPARE", signal13 := "BK23"."X15-2.SPARE", signal14 := "BK23"."X16-2.SPARE", signal15 := "BK23"."X17-2.SPARE", interfaceSignals := #statInterfaceSignalsHmi[26].valueSymbolLeft)
      #instSignals26Right(signal00 :=, signal01 :=, signal02 :=, signal03 :=, signal04 :=, signal05 :=, signal06 :=, signal07 :=, signal08 :=, signal09 :=, signal10 :=, signal11 :=, signal12 :=, signal13 :=, signal14 :=, signal15 :=, interfaceSignals := #statInterfaceSignalsHmi[26].valueSymbolRight)
   END_RUNG
   // the same network as SCL:
   #instSignals26Left(signal00 := "BK23"."X10-1.SEPA CLAMP&CUTTER Z-AXIS LIMIT SENSOR(-)",   // "LAF_InterfaceSignalsBool"
                      signal01 := "BK23"."X11-1.SEPA CLAMP&CUTTER Z-AXIS LIMIT SENSOR(+)",
                      signal02 := "BK23"."X12-1.SEPA CUTTER UP",
                      signal03 := "BK23"."X13-1.SPARE",
                      signal04 := "BK23"."X14-1.SPARE",
                      signal05 := "BK23"."X15-1.SPARE",
                      signal06 := "BK23"."X16-1.SEPA DETECT SENSOR",
                      signal07 := "BK23"."X17-1.SPARE",
                      signal08 := "BK23"."X10-2.CLAMP&CUTTER Z-AXIS HOME SENSOR",
                      signal09 := "BK23"."X11-2.SPARE",
                      signal10 := "BK23"."X12-2.SEPA CUTTER DOWN",
                      signal11 := "BK23"."X13-2.SPARE",
                      signal12 := "BK23"."X14-2.SPARE",
                      signal13 := "BK23"."X15-2.SPARE",
                      signal14 := "BK23"."X16-2.SPARE",
                      signal15 := "BK23"."X17-2.SPARE",
                      interfaceSignals := #statInterfaceSignalsHmi[26].valueSymbolLeft,
                      ENO => #_w1);
   IF #_w1 THEN
       #instSignals26Right(interfaceSignals := #statInterfaceSignalsHmi[26].valueSymbolRight);   // "LAF_InterfaceSignalsBool"
   END_IF;
END_REGION

REGION Network 32: Interface Signals 05 -Example: Model Flex-Pro-Line - IN/OUT- / Interface Signals 27
   // Aufruf des Schnittstellen Signal Bausteins Ba-Bereich 4 / Call the interface signals bool blocks of opmode 4
   RUNG wire#powerrail
      #instSignals27Left(signal00 := "BK24"."X10-1.SEPA CLAMP TOP REAR UP", signal01 := "BK24"."X11-1.SPARE", signal02 := "BK24"."X12-1.SEPA CLAMP TOP FRONT UP", signal03 := "BK24"."X13-1.SPARE", signal04 := "BK24"."X14-1.SEPA CLAMP BTM REAR UP", signal05 := "BK24"."X15-1.SPARE", signal06 := "BK24"."X16-1.SEPA CLAMP BTM FRONT UP", signal07 := "BK24"."X17-1.SPARE", signal08 := "BK24"."X10-2.SEPA CLAMP TOP REAR DOWN", signal09 := "BK24"."X11-2.SPARE", signal10 := "BK24"."X12-2.SEPA CLAMP TOP FRONT DOWN", signal11 := "BK24"."X13-2.SPARE", signal12 := "BK24"."X14-2.SEPA CLAMP BTM REAR DOWN", signal13 := "BK24"."X15-2.SPARE", signal14 := "BK24"."X16-2.SEPA CLAMP BTM FRONT DOWN", signal15 := "BK24"."X17-2.SPARE", interfaceSignals := #statInterfaceSignalsHmi[27].valueSymbolLeft)
      #instSignals27Right(signal00 :=, signal01 :=, signal02 :=, signal03 :=, signal04 :=, signal05 :=, signal06 :=, signal07 :=, signal08 :=, signal09 :=, signal10 :=, signal11 :=, signal12 :=, signal13 :=, signal14 :=, signal15 :=, interfaceSignals := #statInterfaceSignalsHmi[27].valueSymbolRight)
   END_RUNG
   // the same network as SCL:
   #instSignals27Left(signal00 := "BK24"."X10-1.SEPA CLAMP TOP REAR UP",   // "LAF_InterfaceSignalsBool"
                      signal01 := "BK24"."X11-1.SPARE",
                      signal02 := "BK24"."X12-1.SEPA CLAMP TOP FRONT UP",
                      signal03 := "BK24"."X13-1.SPARE",
                      signal04 := "BK24"."X14-1.SEPA CLAMP BTM REAR UP",
                      signal05 := "BK24"."X15-1.SPARE",
                      signal06 := "BK24"."X16-1.SEPA CLAMP BTM FRONT UP",
                      signal07 := "BK24"."X17-1.SPARE",
                      signal08 := "BK24"."X10-2.SEPA CLAMP TOP REAR DOWN",
                      signal09 := "BK24"."X11-2.SPARE",
                      signal10 := "BK24"."X12-2.SEPA CLAMP TOP FRONT DOWN",
                      signal11 := "BK24"."X13-2.SPARE",
                      signal12 := "BK24"."X14-2.SEPA CLAMP BTM REAR DOWN",
                      signal13 := "BK24"."X15-2.SPARE",
                      signal14 := "BK24"."X16-2.SEPA CLAMP BTM FRONT DOWN",
                      signal15 := "BK24"."X17-2.SPARE",
                      interfaceSignals := #statInterfaceSignalsHmi[27].valueSymbolLeft,
                      ENO => #_w1);
   IF #_w1 THEN
       #instSignals27Right(interfaceSignals := #statInterfaceSignalsHmi[27].valueSymbolRight);   // "LAF_InterfaceSignalsBool"
   END_IF;
END_REGION

